// TwinCAT 3 PLC project PLC_1
// ProgramVersion: 3.1.0.4
// libraries:
//   CDS_MemMan, 3.3.2.0 (3S - Smart Software Solutions GmbH)
//   Tc2_Standard, * (Beckhoff Automation GmbH)
//   Tc2_System, * (Beckhoff Automation GmbH)
//   Tc3_Interfaces, * (Beckhoff Automation GmbH)
//   Tc3_Module, * (Beckhoff Automation GmbH)
//   Tc2_Utilities,3.3.0.0,Beckhoff Automation GmbH
// project tree:
//   DUTs/ E_CtrlId.TcDUT (not stored)
//   GVLs/ Global.TcGVL, Io.TcGVL
//   POUs/Alarm/ E_AlmClass.TcDUT, E_AlmState.TcDUT, FB_Alm_Man.TcPOU, T_AlmElement.TcDUT, T_Ctrl_Alm.TcDUT
//   POUs/BaseCtrl/ Base_CmdState.TcGVL, Base_Const.TcGVL, E_Mode.TcDUT, FB_CtrlBase.TcPOU, I_CtrlBase.TcIO, T_Ctrl_CIf.TcDUT, T_Ctrl_Class.TcDUT, T_Ctrl_Class_Alm.TcDUT, T_Ctrl_Class_StateMachine.TcDUT, T_Ctrl_CmdListElement.TcDUT, T_Ctrl_Info.TcDUT, T_Ctrl_IoBool.TcDUT, T_Ctrl_Job.TcDUT, T_Ctrl_SwCfg.TcDUT, T_fbInfo.TcDUT
//   POUs/Controller/Lvl0/CYL/ CYL_CmdState.TcGVL, E_Typ_CYL.TcDUT, FB_CYL.TcPOU, T_Ctrl_SIf_CYL.TcDUT, T_Ctrl_SIf_CYL_Cfg.TcDUT, T_Ctrl_SIf_CYL_Cur.TcDUT, T_Ctrl_SIf_CYL_Ilk.TcDUT (not stored), T_Ctrl_SIf_CYL_In.TcDUT, T_Ctrl_SIf_CYL_Out.TcDUT, T_Ctrl_SIf_CYL_Par.TcDUT
//   POUs/Controller/Lvl2/MOD/ E_Typ_MOD.TcDUT, FB_MOD.TcPOU, MOD_CmdState.TcGVL, T_Ctrl_SIf_MOD.TcDUT, T_Ctrl_SIf_MOD_Cfg.TcDUT (not stored), T_Ctrl_SIf_MOD_Cur.TcDUT, T_Ctrl_SIf_MOD_Ilk.TcDUT, T_Ctrl_SIf_MOD_Par.TcDUT (not stored), T_MOD_RUN_StateMachine.TcDUT (not stored)
//   POUs/Program/ FastPRG_1.TcPOU (not stored), MiddlePRG_1.TcPOU, SlowPRG_1.TcPOU
//   POUs/Utility Functions/ getInBol.TcPOU, getStrInstanceName.TcPOU, setOutBol.TcPOU
//   / Task_Fast.TcTTO, Task_Middle.TcTTO, Task_Slow.TcTTO

CONFIGURATION PLC_1
    RESOURCE PLC ON TwinCAT3
        TASK Task_Fast(INTERVAL := T#10ms, PRIORITY := 5);
        TASK Task_Middle(INTERVAL := T#50000us, PRIORITY := 10);
        TASK Task_Slow(INTERVAL := T#100000us, PRIORITY := 20);
        PROGRAM FastPRG_1 WITH Task_Fast : FastPRG_1;
        PROGRAM MiddlePRG_1 WITH Task_Middle : MiddlePRG_1;
        PROGRAM SlowPRG_1 WITH Task_Slow : SlowPRG_1;
    END_RESOURCE
END_CONFIGURATION

// ---- POUs/Alarm/E_AlmClass.TcDUT
TYPE E_AlmClass :
(
	///no alarm active
	NONE := 0,
	///info
	INFO,
	///warning
	WARNING,
	///tact stop
	TSTOP,
	///stop
	STOP,
	///off
	OFF,
	///Emergency off
	EOFF,
	Max_E_AlmClass
);
END_TYPE

// ---- POUs/Alarm/E_AlmState.TcDUT
TYPE E_AlmState :
(
	///no alarm active
	NONE := 0,
	///alarm clear entry -> set bit1
	CLR := 1,
	///entry resettable alarm ->  set bit2
	RST := 2,
	///entry non resettable alarm ->  set bit2 + bit3
	SET := 3,
	Max_E_AlmState
);
END_TYPE

// ---- POUs/Alarm/T_AlmElement.TcDUT
TYPE T_AlmElement :
STRUCT
	///unique alarm number := 100000*udiMachineNr + intCtrlId*100 + udiAlarmNr
	udiNr: UDINT;
	///additional information - better string???
	dinInfo: DINT;
	///corresponding alarm class
	eClass: E_AlmClass;
	///clear, resetable
	intState: E_AlmState;
	///entry time
	strDTEntry: STRING;
	///from machine (standard = 1)
	udiMachineNr: UDINT;
	///from controller
	intCtrlId: INT;
	///local alarm number
	udiAlarmNr: UDINT;
END_STRUCT
END_TYPE

// ---- POUs/Alarm/T_Ctrl_Alm.TcDUT
TYPE T_Ctrl_Alm :
STRUCT
	///alarm flag array
	bol: BOOL;
	eAlmClass: E_AlmClass;
	strText: STRING;
END_STRUCT
END_TYPE

// ---- POUs/BaseCtrl/E_Mode.TcDUT
{attribute 'qualified_only' := ''}
TYPE E_Mode :
(
	INITIALIZED := 0,
	AUTO := 10,
	SEMI := 11,
	MANU := 12
);
END_TYPE

// ---- POUs/BaseCtrl/T_Ctrl_CIf.TcDUT
TYPE T_Ctrl_CIf :
STRUCT
	Job: T_Ctrl_Job;
	Info: T_Ctrl_Info;
	SwCfg: T_Ctrl_SwCfg;
END_STRUCT
END_TYPE

// ---- POUs/BaseCtrl/T_Ctrl_Class.TcDUT
TYPE T_Ctrl_Class :
STRUCT
	///local test flag to supress cyclic run (for debugging after init)
	bolActivate: BOOL;
	intCmd: INT;
	intCmdLast: INT;
	eModeHistory: E_Mode;
	///local flag mode change detected
	bolChangeBackToAUTO: BOOL;
	StateMachine: T_Ctrl_Class_StateMachine;
	Alarm: T_Ctrl_Class_Alm;
	FUBInfo: T_fbInfo;
END_STRUCT
END_TYPE

// ---- POUs/BaseCtrl/T_Ctrl_Class_Alm.TcDUT
TYPE T_Ctrl_Class_Alm :
STRUCT
	bolResetOk: BOOL;
	///flag positive check me alarm from child
	bolfp: BOOL;
	///local activ alarm class of parent ctrl
	eParent_ActivAlmClass: E_AlmClass;
	///highest local activ alarm class
	eActivAlmClass: E_AlmClass;
END_STRUCT
END_TYPE

// ---- POUs/BaseCtrl/T_Ctrl_Class_StateMachine.TcDUT
TYPE T_Ctrl_Class_StateMachine :
STRUCT
	///actual state
	intState: INT;
	///state of last cycle
	intStateLastCycle: INT;
	///save history backup p.e. in ERROR state
	intStateHistory: INT;
	///set state for next cycle
	intStateNext: INT;
	///[ms] to simulate state in SINGLE_ANSWER
	udiStateSimSetTime_ms: UDINT := 1000;
	///[ms] time in one state
	udiTimeInState_ms: UDINT;
END_STRUCT
END_TYPE

// ---- POUs/BaseCtrl/T_Ctrl_CmdListElement.TcDUT
TYPE T_Ctrl_CmdListElement :
STRUCT
	///command implemented in controller
	intCmd: INT;
	///command is available info for UI
	bolAvailable: BOOL;
	
	// Name of command. Important for UI.
	strName: STRING;
END_STRUCT
END_TYPE

// ---- POUs/BaseCtrl/T_Ctrl_Info.TcDUT
TYPE T_Ctrl_Info :
STRUCT
	///name of controller instance
	strName: STRING(80);
	///class of controller
	strType: STRING(80);
	///unique controller instance identification number
	intCtrlId: INT;
	///unique identification number of parent controller instance
	intParentCtrlId: INT;
	///all inputs valid -> init done
	bolInitDone: BOOL;
	///Childs
	p_afbChild: ARRAY[0..Base_Const.cMaxNrOfChilds] OF POINTER TO BYTE;
	///common interface array of childs
	p_aCIf: ARRAY[0..Base_Const.cMaxNrOfChilds] OF POINTER TO T_Ctrl_CIf;
END_STRUCT
END_TYPE

// ---- POUs/BaseCtrl/T_Ctrl_IoBool.TcDUT
TYPE T_Ctrl_IoBool :
STRUCT
	///mapped io variable to hardware
	map: BOOL;
	///shows the state of (input: mapped, output: set by programm respectiv at the moment one cycle later evtl. from the forcing if forcing active) -> necessary for what?
	state: BOOL;
	///variabel to/ from program
	intern: BOOL;
	///variabel set from UI
	force: BOOL;
	///enable force of single io-datapoint
	EnForce: BOOL;
END_STRUCT
END_TYPE

// ---- POUs/BaseCtrl/T_Ctrl_Job.TcDUT
TYPE T_Ctrl_Job :
STRUCT
	///mode if mode = AUTO -> ACmd will be used, otherwise the MCmd channel is open
	eMode: E_Mode;
	///automatic command from parent ctrl
	intACmd: INT;
	///manual command from UI p.e.
	intMCmd: INT;
	///active cmd
	strCmd: STRING;
	///active state
	intState: INT;
	strState: STRING;
	///if used - show substates for debugging
	strSubState: STRING;
	///event channel to signal special events to parent parallel to status
	intEvt: INT;
	///reset all alarms
	bolAlmReset: BOOL;
	///activate io-forcing
	bolIoForce: BOOL;
	///overwrite suspend all interlocks (for debugging/testing)
	bolIlkOverwrite: BOOL;
	///activ alarm class of parent ctrl
	eParent_ActivAlmClass: E_AlmClass;
	///activ alarm class of me ctrl
	eMe_ActivAlmClass: E_AlmClass;
	///list of all implemented commands
	aCmdList: ARRAY[0..cMaxCmdPerCtrl] OF T_Ctrl_CmdListElement;
END_STRUCT
END_TYPE

// ---- POUs/BaseCtrl/T_Ctrl_SwCfg.TcDUT
TYPE T_Ctrl_SwCfg :
STRUCT
	///hardware/controller exists
	bolExist: BOOL;
	///enable statemachine
	bolEnable: BOOL;
	///set controller in simulation(statemachine active, io local simulated)
	bolSimulation: BOOL;
END_STRUCT
END_TYPE

// ---- POUs/BaseCtrl/T_fbInfo.TcDUT
TYPE T_fbInfo :
STRUCT
	udiSample_ms: UDINT;
END_STRUCT
END_TYPE

// ---- POUs/Controller/Lvl0/CYL/E_Typ_CYL.TcDUT
TYPE E_Typ_CYL :
(
	///bistabile and two feedback sensors
	Valve2_Sensor2 := 0,
	///bistabile and extended feedback sensors	
	Valve2_SensorExtended,
	///bistabile and retracted feedback sensors	
	Valve2_SensorRetracted,
	///bistabile and no feedback sensors
	Valve2_Sensor0,
	///monostabile and 2 feedback sensors	
	Valve1_Sensor2,
	///monostabile and extended feedback sensors	
	Valve1_SensorExtended,
	///monostabile and retracted feedback sensor
	Valve1_SensorRetracted,
	///monostabile and no feedback sensors
	Valve1_Sensor0,
	Max_E_Typ_CYL
);
END_TYPE

// ---- POUs/Controller/Lvl0/CYL/T_Ctrl_SIf_CYL.TcDUT
TYPE T_Ctrl_SIf_CYL :
STRUCT
	///configuration
	Cfg: T_Ctrl_SIf_CYL_Cfg;
	///parameter
	Par: T_Ctrl_SIf_CYL_Par;
	///current values
	Cur: T_Ctrl_SIf_CYL_Cur;
	///io input
	In: T_Ctrl_SIf_CYL_In;
	///io output
	Out: T_Ctrl_SIf_CYL_Out;
	///alarm number used in this controller
	Alm: ARRAY[1..6] OF T_Ctrl_Alm;
	///interlock of output/movements
	Ilk: T_Ctrl_SIf_CYL_Ilk;
END_STRUCT
END_TYPE

// ---- POUs/Controller/Lvl0/CYL/T_Ctrl_SIf_CYL_Cfg.TcDUT
TYPE T_Ctrl_SIf_CYL_Cfg :
STRUCT
	eTyp: E_Typ_CYL;
END_STRUCT
END_TYPE

// ---- POUs/Controller/Lvl0/CYL/T_Ctrl_SIf_CYL_Cur.TcDUT
TYPE T_Ctrl_SIf_CYL_Cur :
STRUCT
	///[ms] time last movement to retract
	udiMoveTimeRetract: UDINT;
	///[ms] time last movement to extend
	udiMoveTimeExtend: UDINT;
END_STRUCT
END_TYPE

// ---- POUs/Controller/Lvl0/CYL/T_Ctrl_SIf_CYL_In.TcDUT
TYPE T_Ctrl_SIf_CYL_In :
STRUCT
	///sensor feedback position extended reached
	bolExtended: T_Ctrl_IoBool;
	///sensor feedback position retracted reached
	bolRetracted: T_Ctrl_IoBool;
END_STRUCT
END_TYPE

// ---- POUs/Controller/Lvl0/CYL/T_Ctrl_SIf_CYL_Out.TcDUT
TYPE T_Ctrl_SIf_CYL_Out :
STRUCT
	///switch valve retract
	bolRetract: T_Ctrl_IoBool;
	///switch valve extend
	bolExtend: T_Ctrl_IoBool;
END_STRUCT
END_TYPE

// ---- POUs/Controller/Lvl0/CYL/T_Ctrl_SIf_CYL_Par.TcDUT
TYPE T_Ctrl_SIf_CYL_Par :
STRUCT
	///[ms] until failure to long time for extend
	udiExtendTime_ms: UDINT;
	///[ms] until failure to long time for retract
	udiRetractTime_ms: UDINT;
	///[ms] simulation time for extend or /2 of timeout time?
	udiSimExtendTime_ms: UDINT;
	///[ms] simulation time for retract or /2 of timeout time?
	udiSimRetractTime_ms: UDINT;
END_STRUCT
END_TYPE

// ---- POUs/Controller/Lvl2/MOD/E_Typ_MOD.TcDUT
TYPE E_Typ_MOD :
(
	///no usage until yet
	Default := 0,
	Max_E_Typ_CYL
);
END_TYPE

// ---- POUs/Controller/Lvl2/MOD/T_Ctrl_SIf_MOD.TcDUT
TYPE T_Ctrl_SIf_MOD :
STRUCT
	///configuration
	Cfg: T_Ctrl_SIf_MOD_Cfg;
	///parameter
	Par: T_Ctrl_SIf_MOD_Par;
	///current values
	Cur: T_Ctrl_SIf_MOD_Cur;
	///In: T_Ctrl_SIf_MOD_In;
	///Out: T_Ctrl_SIf_MOD_Out;
	Alm: ARRAY[1..6] OF T_Ctrl_Alm;
END_STRUCT
END_TYPE

// ---- POUs/Controller/Lvl2/MOD/T_Ctrl_SIf_MOD_Cur.TcDUT
TYPE T_Ctrl_SIf_MOD_Cur :
STRUCT
	///[ms] time last cycle
	udiCycleTime_ms: UDINT;
END_STRUCT
END_TYPE

// ---- POUs/Controller/Lvl2/MOD/T_Ctrl_SIf_MOD_Ilk.TcDUT
TYPE T_Ctrl_SIf_MOD_Ilk :
STRUCT
	///interlock retraction of cylinder
	bolRetract: BOOL;
	///interlock extend of cylinder
	bolExtend: BOOL;
END_STRUCT
END_TYPE

// ---- GVLs/Global.TcGVL
VAR_GLOBAL
	g_a_pCtrlInst: ARRAY[0..E_CtrlId.E_CtrlIdMax] OF POINTER TO fb_CtrlBase;
	g_a_pCtrlCIf: ARRAY[0..E_CtrlId.E_CtrlIdMax] OF POINTER TO T_Ctrl_CIf;
	g_fbAlm_Man: FB_Alm_Man;
END_VAR

// ---- GVLs/Io.TcGVL
VAR_GLOBAL
	///input fb instance Cyl_AB position retract normally open
	In_bolCyl_AB_Retracted_NO: BOOL;
	///input fb instance Cyl_AB position extend normally closed
	In_bolCyl_AB_Extended_NC: BOOL;
	///output fb instance Cyl_AB valve retract
	Out_bolCyl_AB_Retract: BOOL;
	///output fb instance Cyl_AB valve extend
	Out_bolCyl_AB_Extend: BOOL;
END_VAR

// ---- POUs/BaseCtrl/Base_CmdState.TcGVL
VAR_GLOBAL CONSTANT
	///ctrl commands definitions
	///general commands 2-200 - every command has to be a even number
	cCMD_DONE: INT := -1;
	cCMD_INITIALIZED: INT := 0;
	cCMD_PON: INT := 2;
	cCMD_EOFF: INT := 4;
	cCMD_OFF: INT := 6;
	cCMD_INIT: INT := 8;
	cCMD_RUN: INT := 10;
	cCMD_STOP: INT := 12;
	cCMD_TSTOP: INT := 14;
	///ctrl states definitions
	cSTA_DONE: INT := cCMD_DONE;
	cSTA_INITIALIZED: INT := cCMD_INITIALIZED;
	cSTA_PONBusy: INT := 1;
	cSTA_PON: INT := cCMD_PON;
	cSTA_EOFFBusy: INT := 3;
	cSTA_EOFF: INT := cCMD_EOFF;
	cSTA_OFFBusy: INT := 5;
	cSTA_OFF: INT := cCMD_OFF;
	cSTA_INITBusy: INT := 7;
	cSTA_INIT: INT := cCMD_INIT;
	cSTA_RUNBusy: INT := 9;
	cSTA_RUN: INT := cCMD_RUN;
	cSTA_STOPBusy: INT := 11;
	cSTA_STOP: INT := cCMD_STOP;
	cSTA_TSTOPBusy: INT := 13;
	cSTA_TSTOP: INT := cCMD_TSTOP;
	///special states without corresponding cmd
	cSTA_ERROR: INT := 150;
	cSTA_ERRORQuit: INT := 151;
	cSTA_SINGLE_ANSWER: INT := 152;
END_VAR

// ---- POUs/BaseCtrl/Base_Const.TcGVL
VAR_GLOBAL CONSTANT
	///number of child access possible in one controller class
	cMaxNrOfChilds: UINT := 10;
	///maximal number of commands implemented in one controller class
	cMaxCmdPerCtrl: UINT := 15;
	///maximal number of commands implemented in one controller class
	cMaxBaseCmdState: UINT := 200;
END_VAR

// ---- POUs/Controller/Lvl0/CYL/CYL_CmdState.TcGVL
VAR_GLOBAL CONSTANT
	///ctrl commands definitions
	///specific commands >200 - every command has to be a even number
	cCMD_RETRACT: INT := 202;
	cCMD_EXTEND: INT := 204;
	///ctrl specific states definitions
	cSTA_RETRACTBusy: INT := 201;
	cSTA_RETRACT: INT := cCMD_RETRACT;
	cSTA_EXTENDBusy: INT := 203;
	cSTA_EXTEND: INT := cCMD_EXTEND;
END_VAR

// ---- POUs/Controller/Lvl2/MOD/MOD_CmdState.TcGVL
VAR_GLOBAL CONSTANT
	///ctrl commands definitions
	///specific commands >200 - every command has to be a even number
	///ctrl specific states definitions
	cSTA_VER_Up: INT := 201;
	cSTA_VER_Down: INT := 202;
	cSTA_WAIT_Pick: INT := 203;
	cSTA_HOR_MoveToPlace: INT := 204;
	cSTA_HOR_MoveToPick: INT := 205;
	cSTA_Finished: INT := 206;
END_VAR

// ---- POUs/BaseCtrl/I_CtrlBase.TcIO
INTERFACE I_CtrlBase

METHOD iniCtrlArray : BOOL
VAR_INPUT
	p_pCtrlArray: POINTER TO POINTER TO fb_CtrlBase;
	intCtrlID: INT;
END_VAR
END_METHOD

METHOD getCtrlCIf : POINTER TO T_Ctrl_CIf
END_METHOD

END_INTERFACE

// ---- POUs/Program/MiddlePRG_1.TcPOU
PROGRAM MiddlePRG_1
VAR
	bolPlcStartupDone: BOOL := FALSE;
	bolHostInitDone : BOOL := FALSE;
	bolInitDone : BOOL := FALSE;
	fbCyl_AB: FB_CYL;
	fbMOD_2: FB_MOD;
	fbVER_2: FB_CYL;
	fbHOR_2: FB_CYL;
END_VAR

(*__________________________________________________________________________________________________
¦	
¦	Vistaprint Schweiz GmbH
¦	CH - 8401 Winterthur
¦
¦	www.vistaprint.ch - info@vistaprint.ch
¦___________________________________________________________________________________________________

Function desription:
call of all controller (FUB) for the middel task class inclusiv alarm handler.


History:
Version		Date			Author		Comment
---------------------------------------------------------------------------------------------------
0.00.1		02.05.2013		AVME/KVO	Start history


___________________________________________________________________________________________________*)

// -----------------------------------------------------------------------------------------------
// Initialize the PLC Parameter and check the PLC health
// -----------------------------------------------------------------------------------------------
IF (NOT bolPlcStartupDone) THEN
	bolPlcStartupDone := TRUE;	
END_IF
// -----------------------------------------------------------------------------------------------


// -----------------------------------------------------------------------------------------------
// The host system is downloading all parameter at startup. 
// bolPlcStartupDone will be set to true after the Host is done with the initialization
// -----------------------------------------------------------------------------------------------
IF (bolPlcStartupDone AND (NOT bolHostInitDone) AND NOT bolInitDone) THEN
	bolHostInitDone := TRUE;
END_IF
// -----------------------------------------------------------------------------------------------


// -----------------------------------------------------------------------------------------------
// Start PLC code initialization
// -----------------------------------------------------------------------------------------------
IF NOT bolInitDone AND bolPlcStartupDone AND bolHostInitDone THEN
	
	// init
	fbCyl_AB.iniCtrlArray(ADR(g_a_pCtrlInst),E_CtrlId.CYL_VER1);     	// init and entry fb_instance in global fb pointer array
	g_a_pCtrlCIf[E_CtrlId.CYL_VER1] := fbCyl_AB.getCtrlCIf();    // get adr of ctrl interface struct
	
	// init module example
	// Lvl0
	fbHOR_2.iniCtrlArray(ADR(g_a_pCtrlInst),E_CtrlId.HOR_2); // init and entry fb_instance in global fb pointer array
	g_a_pCtrlCIf[E_CtrlId.HOR_2] := fbHOR_2.getCtrlCIf();    // get adr of ctrl interface struct
	
	fbVER_2.iniCtrlArray(ADR(g_a_pCtrlInst),E_CtrlId.VER_2); // init and entry fb_instance in global fb pointer array
	g_a_pCtrlCIf[E_CtrlId.VER_2] := fbVER_2.getCtrlCIf();    // get adr of ctrl interface struct
	
	//Lvl2
	fbMOD_2.iniCtrlArray(ADR(g_a_pCtrlInst),E_CtrlId.MOD_2); // init and entry fb_instance in global fb pointer array
	g_a_pCtrlCIf[E_CtrlId.MOD_2] := fbMOD_2.getCtrlCIf();    // get adr of ctrl interface struct
	
	// add childs
	fbMOD_2.p_fbHOR := g_a_pCtrlInst[E_CtrlId.HOR_2];
	fbMOD_2.p_fbVER := g_a_pCtrlInst[E_CtrlId.VER_2];

	// add childs
	fbMOD_2.p_fbHOR := g_a_pCtrlInst[E_CtrlId.HOR_2];
	fbMOD_2.p_fbVER := g_a_pCtrlInst[E_CtrlId.VER_2];

	bolInitDone := TRUE;
END_IF
// -----------------------------------------------------------------------------------------------



// -----------------------------------------------------------------------------------------------
// Normal Run mode after all the initialization is done
// -----------------------------------------------------------------------------------------------
IF (bolInitDone AND bolPlcStartupDone AND bolHostInitDone) THEN
	
	//****************************************************************************************************
	// cyclic controller calls
	//****************************************************************************************************
	fbCyl_AB.In_bolRetracted := In_bolCyl_AB_Retracted_NO;
	fbCyl_AB.In_bolExtended := (NOT In_bolCyl_AB_Extended_NC);
	fbCyl_AB();
	Out_bolCyl_AB_Retract := fbCyl_AB.Out_bolRetract;
	Out_bolCyl_AB_Extend := fbCyl_AB.Out_bolExtend;

	// Modul example
	// ----------------------------------------------------------------------------------------------------------------------------
	// modul controller MOD_2 with childs
	fbMOD_2();
	fbVER_2();
	fbHOR_2();

	
END_IF
// -----------------------------------------------------------------------------------------------

END_PROGRAM

// ---- POUs/Controller/Lvl0/CYL/FB_CYL.TcPOU
FUNCTION_BLOCK FB_CYL EXTENDS FB_CtrlBase

VAR_INPUT
	In_bolRetracted: BOOL;
	In_bolExtended: BOOL;
END_VAR
VAR_OUTPUT
	Out_bolRetract: BOOL;
	Out_bolExtend: BOOL;
END_VAR

VAR
	/// Specific interface struct for public access
	SIf: T_Ctrl_SIf_CYL;
	
END_VAR

(*__________________________________________________________________________________________________
¦	
¦	Vistaprint Schweiz GmbH
¦	CH - 8401 Winterthur
¦
¦	www.vistaprint.ch - info@vistaprint.ch
¦___________________________________________________________________________________________________

Function desription:
Basic controller implementation. This Controller should be the base father controller for all in the
feature implemented ctontroller classes.


History:
Version		Date			Author		Comment
---------------------------------------------------------------------------------------------------
0.00.1		25.04.2013		AVME/KVO	Start history


___________________________________________________________________________________________________*)


IF (me.bolActivate) THEN // cyclic call enabled
	IF (CIf.Info.bolInitDone=FALSE) THEN // first cycle -> init
		CtrlInit();
		CIf.Info.bolInitDone := TRUE;
	ELSE
		CycleStartDuty();
	
		Always();
		
		StateMachine();
		
		CycleEndDuty();
	END_IF
END_IF;

METHOD FB_init : BOOL
VAR_INPUT
	///if TRUE, the retain variables are initialized (warm start / cold start)
	bInitRetains: BOOL;
	///if TRUE, the instance afterwards gets moved into the copy code (online change)
	bInCopyCode: BOOL;
END_VAR
VAR
	udiTaskCnt: UDINT;
	ii: UINT;
END_VAR
//------------------------------------------------------------------------------------------------------------------------
// to manually change in new FUB implementation!!!
// define valid commands for this controller
FOR ii:= 0 TO (SIZEOF(CIf.Job.aCmdList)/SIZEOF(CIf.Job.aCmdList[0])-1) BY 1 DO
	IF (CIf.Job.aCmdList[ii].intCmd=cCMD_INITIALIZED) THEN
		// found first empty array element
		EXIT;
	END_IF
END_FOR
CIf.Job.aCmdList[ii].intCmd := cCMD_STOP;
CIf.Job.aCmdList[ii].strName := 'Stop'; 
CIf.Job.aCmdList[ii].bolAvailable := TRUE;
ii := ii +1;
CIf.Job.aCmdList[ii].intCmd := cCMD_RETRACT;
CIf.Job.aCmdList[ii].strName := 'Retract';
CIf.Job.aCmdList[ii].bolAvailable := TRUE;
ii := ii +1;
CIf.Job.aCmdList[ii].intCmd := cCMD_EXTEND; // for test simulation single answer
CIf.Job.aCmdList[ii].strName := 'Extend';
CIf.Job.aCmdList[ii].bolAvailable := TRUE;

// set name of class/typ
CIf.Info.strType := 'FB_CYL'; 

// set alarm class
SIf.Alm[1].eAlmClass := E_AlmClass.EOFF;
//SIf.Alm[1].strAlarm := 'Alarmtext 1';
SIf.Alm[2].eAlmClass := E_AlmClass.OFF;
SIf.Alm[3].eAlmClass := E_AlmClass.STOP;
SIf.Alm[4].eAlmClass := E_AlmClass.TSTOP;
SIf.Alm[5].eAlmClass := E_AlmClass.INFO;
SIf.Alm[6].eAlmClass := E_AlmClass.WARNING;

//*******************************************************************************
// initial values
//*******************************************************************************

// software configuration
CIf.SwCfg.bolExist := TRUE;
CIf.SwCfg.bolSimulation := TRUE;

// parmeter
SIf.Par.udiExtendTime_ms := 10000;
SIf.Par.udiRetractTime_ms := 8000;
SIf.Par.udiSimExtendTime_ms := SIf.Par.udiExtendTime_ms/2;	
SIf.Par.udiSimRetractTime_ms := SIf.Par.udiRetractTime_ms/2;
END_METHOD

METHOD PROTECTED IoInBridge : BOOL
// digitale and analoge inputs read from hardware or forcing
SIf.In.bolExtended.map := THIS^.In_bolExtended;
SIf.In.bolRetracted.map := THIS^.In_bolRetracted;

IF (CIf.SwCfg.bolSimulation = FALSE) THEN
	getInBol(CIf.Job.bolIoForce,ADR(SIf.In.bolExtended));
	getInBol(CIf.Job.bolIoForce,ADR(SIf.In.bolRetracted));
	//ctrl.In.bol_PosSwitchBasicDefTyp.intern := getInBol(ctrl.ifc.Job.bol_Force ,ADR(ctrl.In.bol_PosSwitchBasicDefTyp);
ELSE
	//simulation of global IO
END_IF
END_METHOD

METHOD PROTECTED IoOutBridge : BOOL
VAR
	bolSwitchValvesOff: BOOL;
END_VAR
// digitale and analoge inputs read from hardware or forcing
IF (CIf.SwCfg.bolSimulation = FALSE) THEN
	// check interlocks to prevent damages
	IF (CIf.Job.bolIlkOverwrite=FALSE) THEN
		bolSwitchValvesOff := FALSE;
		
		IF (SIf.Ilk.bolExtend=FALSE) THEN
			setOutBol(CIf.Job.bolIoForce ,ADR(SIf.Out.bolExtend));
		ELSE
			// switch off?
			IF (SIf.Cfg.eTyp = E_Typ_CYL.Valve1_Sensor0) OR (SIf.Cfg.eTyp = E_Typ_CYL.Valve1_Sensor2) 
				OR (SIf.Cfg.eTyp = E_Typ_CYL.Valve1_SensorExtended) OR (SIf.Cfg.eTyp = E_Typ_CYL.Valve1_SensorRetracted) THEN
				// monostabil valve -> do nothing
			ELSE
				// bistable valve ->  switch both off
				bolSwitchValvesOff := TRUE;
			END_IF
		END_IF
		
		IF (SIf.Ilk.bolRetract=FALSE) THEN
			setOutBol(CIf.Job.bolIoForce ,ADR(SIf.Out.bolRetract));
		ELSE
			// switch off?
			IF (SIf.Cfg.eTyp = E_Typ_CYL.Valve1_Sensor0) OR (SIf.Cfg.eTyp = E_Typ_CYL.Valve1_Sensor2) 
				OR (SIf.Cfg.eTyp = E_Typ_CYL.Valve1_SensorExtended) OR (SIf.Cfg.eTyp = E_Typ_CYL.Valve1_SensorRetracted) THEN
				// monostabil valve -> do nothing
				;
			ELSE
				// bistable valve -> switch both off
				bolSwitchValvesOff := TRUE;
			END_IF
		END_IF
		
		// bistable valve -> switch both off
		IF (bolSwitchValvesOff) THEN
			SIf.Out.bolExtend.map := FALSE;
			SIf.Out.bolRetract.map := FALSE;
		END_IF
		
	END_IF
END_IF
END_METHOD

METHOD PROTECTED StateMachine : BOOL
SUPER^.StateMachine();

// main statemachine of base controller
CASE me.StateMachine.intState OF
    cSTA_RETRACTBusy: 
        THIS^.sta_RETRACTBusy();
    cSTA_RETRACT: 
        THIS^.sta_RETRACT();
    cSTA_EXTENDBusy: 
        THIS^.sta_EXTENDBusy();
    cSTA_EXTEND: 
        THIS^.sta_EXTEND();
END_CASE;
END_METHOD

METHOD PROTECTED sta_ERROR : BOOL
// state implemetation
//--------------------------------------------------------------------------------------
// Entry action
	IF (me.StateMachine.intState<>me.StateMachine.intStateHistory) THEN
		me.StateMachine.intStateHistory := me.StateMachine.intStateLastCycle; // -> possibillity to go back to state before error
		me.StateMachine.intStateLastCycle := me.StateMachine.intState;
		
	END_IF


//--------------------------------------------------------------------------------------
// Cyclic action
	IF (me.StateMachine.intState=me.StateMachine.intStateLastCycle) THEN
		
		;
		
		
		// State Change Condition
		IF (CIf.Job.bolAlmReset = TRUE) THEN
			me.StateMachine.intStateNext := cSTA_ERRORQuit;
		END_IF
	END_IF




//--------------------------------------------------------------------------------------
// Exit action
	IF (me.StateMachine.intState<>me.StateMachine.intStateNext) THEN
		;
	END_IF
END_METHOD

METHOD PROTECTED sta_ERRORQuit : BOOL
// state implemetation
//--------------------------------------------------------------------------------------
// Entry action
	IF (me.StateMachine.intState<>me.StateMachine.intStateLastCycle) THEN
		me.StateMachine.intStateLastCycle := me.StateMachine.intState;
		
	END_IF


//--------------------------------------------------------------------------------------
// Cyclic action
	IF (me.StateMachine.intState=me.StateMachine.intStateLastCycle) THEN
		
		;
		// evtl. wait time if reset of device is necessary and then decide to go to states or ERROR state
		IF (CIf.Job.bolAlmReset = TRUE) THEN
			CIf.Job.eMe_ActivAlmClass := E_AlmClass.NONE; // reset feedback channel for parent
			CIf.Job.bolAlmReset := FALSE;
		END_IF
		
		// State Change Condition
		IF (CIf.Job.bolAlmReset = FALSE) THEN
			IF (me.StateMachine.intStateHistory<=cSTA_PON) THEN
				me.StateMachine.intStateNext := cSTA_PONBusy;
			ELSIF(me.intCmd=cCMD_OFF) THEN
				me.StateMachine.intStateNext := cSTA_OFFBusy;
			ELSIF(me.intCmd=cCMD_STOP) THEN
				me.StateMachine.intStateNext := cSTA_STOPBusy;
			ELSIF(me.intCmd=cCMD_RETRACT) THEN
				me.StateMachine.intStateNext := cSTA_RETRACTBusy;
			ELSIF(me.intCmd=cCMD_EXTEND) THEN
				me.StateMachine.intStateNext := cSTA_EXTENDBusy;
			END_IF
		END_IF
	END_IF




//--------------------------------------------------------------------------------------
// Exit action
	IF (me.StateMachine.intState<>me.StateMachine.intStateNext) THEN
		;
	END_IF
END_METHOD

METHOD PROTECTED sta_EXTENDBusy : BOOL
// state implemetation
//--------------------------------------------------------------------------------------
// Entry action
	IF (me.StateMachine.intState<>me.StateMachine.intStateLastCycle) THEN
		me.StateMachine.intStateLastCycle := me.StateMachine.intState;

		fbSimulationTimer.IN := FALSE;
		fbSimulationTimer.PT := UDINT_TO_TIME(SIf.Par.udiSimExtendTime_ms);
		fbSimulationTimer(); // set time/reset timer
		fbSimulationTimer.IN := TRUE; // start timer
	END_IF


//--------------------------------------------------------------------------------------
// Cyclic action
	IF (me.StateMachine.intState=me.StateMachine.intStateLastCycle) THEN

		// Simulation
		IF (CIf.SwCfg.bolSimulation) THEN
			fbSimulationTimer(); // simulation time
			IF (fbSimulationTimer.Q) THEN
				SIf.In.bolExtended.intern := TRUE;
				SIf.In.bolRetracted.intern := FALSE;
			END_IF
		END_IF
		
		//no change action
		SIf.Out.bolExtend.intern := TRUE;
		SIf.Out.bolRetract.intern := FALSE;
		
		
		// State Change Condition
		IF (me.StateMachine.udiTimeInState_ms>SIf.Par.udiExtendTime_ms) THEN
			IF (SIf.In.bolRetracted.intern) THEN
				// sensor retract always on cylinder
				g_fbAlm_Man.setAlarm(CIf.Info.intCtrlId,1,777,ADR(SIf.Alm),E_AlmState.RST,CIf.Job.eMe_ActivAlmClass);
			ELSE
				// timeout extend cylinder
				g_fbAlm_Man.setAlarm(CIf.Info.intCtrlId,2,0,ADR(SIf.Alm),E_AlmState.RST,CIf.Job.eMe_ActivAlmClass);
			END_IF
			me.StateMachine.intStateNext :=  cSTA_ERROR;
		ELSIF (SIf.In.bolExtended.intern) AND (SIf.In.bolRetracted.intern=FALSE) THEN
			me.StateMachine.intStateNext := cSTA_EXTEND;
		ELSIF(me.intCmd=cCMD_OFF) THEN
			me.StateMachine.intStateNext := cSTA_OFFBusy;
		ELSIF(me.intCmd=cCMD_STOP) THEN
			me.StateMachine.intStateNext := cSTA_STOPBusy;
		ELSIF(me.intCmd=cCMD_RETRACT) THEN
			me.StateMachine.intStateNext := cSTA_RETRACTBusy;
		END_IF
	END_IF




//--------------------------------------------------------------------------------------
// Exit action
	IF (me.StateMachine.intState<>me.StateMachine.intStateNext) THEN
		SIf.Cur.udiMoveTimeExtend := me.StateMachine.udiTimeInState_ms;
	END_IF
END_METHOD

METHOD PROTECTED sta_EXTEND : BOOL
// state implemetation
//--------------------------------------------------------------------------------------
// Entry action
	IF (me.StateMachine.intState<>me.StateMachine.intStateLastCycle) THEN
		me.StateMachine.intStateLastCycle := me.StateMachine.intState;

	END_IF


//--------------------------------------------------------------------------------------
// Cyclic action
	IF (me.StateMachine.intState=me.StateMachine.intStateLastCycle) THEN

		// Simulation
		IF (CIf.SwCfg.bolSimulation) THEN
			;
		END_IF
		
		// State Change Condition
		IF (SIf.In.bolRetracted.intern) THEN
			// sensor retract always on cylinder
			me.StateMachine.intStateNext :=  cSTA_ERROR;
		ELSIF (SIf.In.bolExtended.intern = FALSE) THEN // wait time until error?
			me.StateMachine.intStateNext := cSTA_EXTENDBusy;
		ELSIF(me.intCmd=cCMD_OFF) THEN
			me.StateMachine.intStateNext := cSTA_OFFBusy;
		ELSIF(me.intCmd=cCMD_STOP) THEN
			me.StateMachine.intStateNext := cSTA_STOPBusy;
		ELSIF(me.intCmd=cCMD_RETRACT) THEN
			me.StateMachine.intStateNext := cSTA_RETRACTBusy;
		END_IF
	END_IF




//--------------------------------------------------------------------------------------
// Exit action
	IF (me.StateMachine.intState<>me.StateMachine.intStateNext) THEN
		;
	END_IF
END_METHOD

METHOD PROTECTED sta_RETRACT : BOOL
// state implemetation
//--------------------------------------------------------------------------------------
// Entry action
	IF (me.StateMachine.intState<>me.StateMachine.intStateLastCycle) THEN
		me.StateMachine.intStateLastCycle := me.StateMachine.intState;

	END_IF


//--------------------------------------------------------------------------------------
// Cyclic action
	IF (me.StateMachine.intState=me.StateMachine.intStateLastCycle) THEN

		// Simulation
		IF (CIf.SwCfg.bolSimulation) THEN
			;
		END_IF
		
		// State Change Condition
		IF (SIf.In.bolExtended.intern) THEN
			// sensor retract always on cylinder
			me.StateMachine.intStateNext :=  cSTA_ERROR;
		ELSIF (SIf.In.bolRetracted.intern = FALSE) THEN // wait time until error?
			me.StateMachine.intStateNext := cSTA_RETRACTBusy;
		ELSIF(me.intCmd=cCMD_OFF) THEN
			me.StateMachine.intStateNext := cSTA_OFFBusy;
		ELSIF(me.intCmd=cCMD_STOP) THEN
			me.StateMachine.intStateNext := cSTA_STOPBusy;
		ELSIF(me.intCmd=cCMD_EXTEND) THEN
			me.StateMachine.intStateNext := cSTA_EXTENDBusy;
		END_IF
	END_IF




//--------------------------------------------------------------------------------------
// Exit action
	IF (me.StateMachine.intState<>me.StateMachine.intStateNext) THEN
		;
	END_IF
END_METHOD

METHOD PROTECTED sta_RETRACTBusy : BOOL
// state implemetation
//--------------------------------------------------------------------------------------
// Entry action
	IF (me.StateMachine.intState<>me.StateMachine.intStateLastCycle) THEN
		me.StateMachine.intStateLastCycle := me.StateMachine.intState;
		
		SIf.Out.bolExtend.intern := FALSE;
		SIf.Out.bolRetract.intern := TRUE;
		
		fbSimulationTimer.IN := FALSE;
		fbSimulationTimer.PT := UDINT_TO_TIME(SIf.Par.udiSimRetractTime_ms);
		fbSimulationTimer(); // set time/reset timer
		fbSimulationTimer.IN := TRUE; // start timer
	END_IF


//--------------------------------------------------------------------------------------
// Cyclic action
	IF (me.StateMachine.intState=me.StateMachine.intStateLastCycle) THEN

		// Simulation
		IF (CIf.SwCfg.bolSimulation) THEN
			fbSimulationTimer(); // simulation time
			IF (fbSimulationTimer.Q) THEN
				SIf.In.bolRetracted.intern := TRUE;
				SIf.In.bolExtended.intern := FALSE;
			END_IF
		END_IF
		
		// State Change Condition
		IF (me.StateMachine.udiTimeInState_ms>SIf.Par.udiRetractTime_ms) THEN
			IF (SIf.In.bolExtended.intern) THEN
				// sensor retract always on cylinder
				g_fbAlm_Man.setAlarm(CIf.Info.intCtrlId,3,0,ADR(SIf.Alm),E_AlmState.RST,CIf.Job.eMe_ActivAlmClass);
			ELSE
				// timeout extend cylinder
				g_fbAlm_Man.setAlarm(CIf.Info.intCtrlId,4,0,ADR(SIf.Alm),E_AlmState.RST,CIf.Job.eMe_ActivAlmClass);
			END_IF
			me.StateMachine.intStateNext :=  cSTA_ERROR;
		ELSIF (SIf.In.bolRetracted.intern) AND(SIf.In.bolExtended.intern=FALSE) THEN
			me.StateMachine.intStateNext := cSTA_RETRACT;
		ELSIF(me.intCmd=cCMD_OFF) THEN
			me.StateMachine.intStateNext := cSTA_OFFBusy;
		ELSIF(me.intCmd=cCMD_STOP) THEN
			me.StateMachine.intStateNext := cSTA_STOPBusy;
		ELSIF(me.intCmd=cCMD_EXTEND) THEN
			me.StateMachine.intStateNext := cSTA_EXTENDBusy;
		END_IF
	END_IF




//--------------------------------------------------------------------------------------
// Exit action
	IF (me.StateMachine.intState<>me.StateMachine.intStateNext) THEN
		SIf.Cur.udiMoveTimeRetract := me.StateMachine.udiTimeInState_ms;
	END_IF
END_METHOD

METHOD getCtrlSIf : POINTER TO T_Ctrl_SIf_CYL
getCtrlSIf := ADR(SIf);
END_METHOD

METHOD PROTECTED sta_PON : BOOL
// state implemetation
//--------------------------------------------------------------------------------------
// Entry action
	IF (me.StateMachine.intState<>me.StateMachine.intStateLastCycle) THEN
		me.StateMachine.intStateLastCycle := me.StateMachine.intState;
		
	END_IF


//--------------------------------------------------------------------------------------
// Cyclic action
	IF (me.StateMachine.intState=me.StateMachine.intStateLastCycle) THEN
		
		;
		
		
		// State Change Condition
		IF(me.intCmd=cCMD_OFF) THEN
			me.StateMachine.intStateNext := cSTA_OFFBusy;
		ELSIF(me.intCmd=cCMD_STOP) THEN
			me.StateMachine.intStateNext := cSTA_STOPBusy;
		ELSIF(me.intCmd=cCMD_RETRACT) THEN
			me.StateMachine.intStateNext := cSTA_RETRACTBusy;
		ELSIF (me.intCmd=cCMD_EXTEND) THEN
			me.StateMachine.intStateNext := cSTA_EXTENDBusy;
		END_IF
	END_IF




//--------------------------------------------------------------------------------------
// Exit action
	IF (me.StateMachine.intState<>me.StateMachine.intStateNext) THEN
		;
	END_IF
END_METHOD

METHOD PROTECTED CtrlInit : BOOL
SUPER^.CtrlInit();
END_METHOD

METHOD PROTECTED getCmdState : STRING
VAR_INPUT
	intCmdState: INT;
	bolState: BOOL;
END_VAR
getCmdState := SUPER^.getCmdState(intCmdState:=intCmdState,bolState:=bolState); // get global/base defined cmds/states
IF (getCmdState='') THEN // global not defined get local
	// get string cmd/state string information in runtime
	IF (bolState=FALSE) THEN
		// cmd's
		CASE intCmdState OF
			cCMD_RETRACT: 
				getCmdState := 'cCMD_RETRACT';
			cCMD_EXTEND: 
				getCmdState := 'cCMD_EXTEND';
		END_CASE;
	ELSE
	
	// cmd's
		CASE intCmdState OF
			cSTA_RETRACTBusy: 
				getCmdState := 'cSTA_RETRACTBusy';
			cSTA_RETRACT: 
				getCmdState := 'cSTA_RETRACT';
			cSTA_EXTENDBusy: 
				getCmdState := 'cSTA_EXTENDBusy';
			cCMD_EXTEND: 
				getCmdState := 'cCMD_EXTEND';
		END_CASE;
	END_IF
END_IF
END_METHOD

METHOD PROTECTED sta_OFF : BOOL
// state implemetation
//--------------------------------------------------------------------------------------
// Entry action
	IF (me.StateMachine.intState<>me.StateMachine.intStateLastCycle) THEN
		me.StateMachine.intStateLastCycle := me.StateMachine.intState;
		
	END_IF


//--------------------------------------------------------------------------------------
// Cyclic action
	IF (me.StateMachine.intState=me.StateMachine.intStateLastCycle) THEN
		
		;
		
		
		// State Change Condition
		IF (me.intCmd=cCMD_STOP) THEN
			// sensor retract always on cylinder
			me.StateMachine.intStateNext :=  cSTA_STOPBusy;
		ELSIF (me.intCmd=cCMD_EXTEND) THEN 
			me.StateMachine.intStateNext := cSTA_EXTENDBusy;
		ELSIF(me.intCmd=cCMD_RETRACT) THEN
			me.StateMachine.intStateNext := cSTA_RETRACTBusy;
		END_IF
	END_IF




//--------------------------------------------------------------------------------------
// Exit action
	IF (me.StateMachine.intState<>me.StateMachine.intStateNext) THEN
		;
	END_IF
END_METHOD

METHOD PROTECTED sta_OFFBusy : BOOL
// state implemetation
//--------------------------------------------------------------------------------------
// Entry action
	IF (me.StateMachine.intState<>me.StateMachine.intStateLastCycle) THEN
		me.StateMachine.intStateLastCycle := me.StateMachine.intState;
		
	END_IF


//--------------------------------------------------------------------------------------
// Cyclic action
	IF (me.StateMachine.intState=me.StateMachine.intStateLastCycle) THEN
		
		// switch off?
		IF (SIf.Cfg.eTyp = E_Typ_CYL.Valve1_Sensor0) OR (SIf.Cfg.eTyp = E_Typ_CYL.Valve1_Sensor2) 
			OR (SIf.Cfg.eTyp = E_Typ_CYL.Valve1_SensorExtended) OR (SIf.Cfg.eTyp = E_Typ_CYL.Valve1_SensorRetracted) THEN
			// monostabil valve -> do nothing
			;
		ELSE
			// bistable valve -> switch both off
			SIf.Out.bolExtend.intern := FALSE;
			SIf.Out.bolRetract.intern := FALSE;
		END_IF
		
		
		
		// State Change Condition
		IF (FALSE) THEN
			;
		ELSIF (TRUE) THEN
			me.StateMachine.intStateNext := cSTA_OFF;
		END_IF
	END_IF




//--------------------------------------------------------------------------------------
// Exit action
	IF (me.StateMachine.intState<>me.StateMachine.intStateNext) THEN
		;
	END_IF
END_METHOD

METHOD PROTECTED sta_STOP : BOOL
// state implemetation
//--------------------------------------------------------------------------------------
// Entry action
	IF (me.StateMachine.intState<>me.StateMachine.intStateLastCycle) THEN
		me.StateMachine.intStateLastCycle := me.StateMachine.intState;
		
	END_IF


//--------------------------------------------------------------------------------------
// Cyclic action
	IF (me.StateMachine.intState=me.StateMachine.intStateLastCycle) THEN
		
		;
		
		
		// State Change Condition
		IF (me.intCmd=cCMD_OFF) THEN
			// sensor retract always on cylinder
			me.StateMachine.intStateNext :=  cSTA_OFFBusy;
		ELSIF (me.intCmd=cCMD_EXTEND) THEN 
			me.StateMachine.intStateNext := cSTA_EXTENDBusy;
		ELSIF(me.intCmd=cCMD_RETRACT) THEN
			me.StateMachine.intStateNext := cSTA_RETRACTBusy;
		END_IF
	END_IF




//--------------------------------------------------------------------------------------
// Exit action
	IF (me.StateMachine.intState<>me.StateMachine.intStateNext) THEN
		;
	END_IF
END_METHOD

METHOD PROTECTED sta_STOPBusy : BOOL
// state implemetation
//--------------------------------------------------------------------------------------
// Entry action
	IF (me.StateMachine.intState<>me.StateMachine.intStateLastCycle) THEN
		me.StateMachine.intStateLastCycle := me.StateMachine.intState;
		
	END_IF


//--------------------------------------------------------------------------------------
// Cyclic action
	IF (me.StateMachine.intState=me.StateMachine.intStateLastCycle) THEN
		
		// switch off?
		IF (SIf.Cfg.eTyp = E_Typ_CYL.Valve1_Sensor0) OR (SIf.Cfg.eTyp = E_Typ_CYL.Valve1_Sensor2) 
			OR (SIf.Cfg.eTyp = E_Typ_CYL.Valve1_SensorExtended) OR (SIf.Cfg.eTyp = E_Typ_CYL.Valve1_SensorRetracted) THEN
			// monostabil valve -> do nothing
			;
		ELSE
			// bistable valve -> switch both on -> block at position
			SIf.Out.bolExtend.intern := TRUE;
			SIf.Out.bolRetract.intern := TRUE;
		END_IF
		
		
		
		// State Change Condition
		IF (FALSE) THEN
			;
		ELSIF (TRUE) THEN
			me.StateMachine.intStateNext := cSTA_STOP;
		END_IF
	END_IF




//--------------------------------------------------------------------------------------
// Exit action
	IF (me.StateMachine.intState<>me.StateMachine.intStateNext) THEN
		;
	END_IF
END_METHOD

END_FUNCTION_BLOCK

// ---- POUs/BaseCtrl/FB_CtrlBase.TcPOU
{attribute 'reflection' := ''}
FUNCTION_BLOCK FB_CtrlBase IMPLEMENTS I_CtrlBase
VAR
	///Commen interface struct for public access
	CIf: T_Ctrl_CIf;
	///basic local controller class struct
	me: T_Ctrl_Class;
	fbSimulationTimer: TON;
	{attribute 'instance-path' := ''}
	{attribute 'noinit' := ''}
	strMyInstancePath: STRING;
END_VAR

(*__________________________________________________________________________________________________
¦	
¦	Vistaprint Schweiz GmbH
¦	CH - 8401 Winterthur
¦
¦	www.vistaprint.ch - info@vistaprint.ch
¦___________________________________________________________________________________________________

Function desription:
Basic controller implementation. This Controller should be the base father controller for all in the
feature implemented ctontroller classes.


History:
Version		Date			Author		Comment
---------------------------------------------------------------------------------------------------
0.00.1		25.04.2013		AVME/KVO	Start history


___________________________________________________________________________________________________*)


IF (me.bolActivate) THEN // cyclic call enabled
	
	IF (CIf.Info.bolInitDone=FALSE) THEN // first cycle -> init
		CtrlInit();
		CIf.Info.bolInitDone := TRUE;
	ELSE
		CycleStartDuty();
	
		Always();
		
		StateMachine();
		
		CycleEndDuty();
	END_IF
	
END_IF;

METHOD iniCtrlArray : BOOL
VAR_INPUT
	p_pCtrlArray: POINTER TO POINTER TO FB_CtrlBase;
	intCtrlID: INT;
END_VAR
iniCtrlArray := FALSE;

IF (TRUE) THEN//e_CtrlID <= E_CtrlId.E_CtrlIdMax) THEN
	p_pCtrlArray[intCtrlID] := THIS;
	THIS^.CIf.Info.intCtrlID := intCtrlID;
	iniCtrlArray := TRUE;
END_IF
END_METHOD

METHOD FB_init : BOOL
VAR_INPUT
	///if TRUE, the retain variables are initialized (warm start / cold start)
	bInitRetains: BOOL;
	///if TRUE, the instance afterwards gets moved into the copy code (online change)
	bInCopyCode: BOOL;
END_VAR
//------------------------------------------------------------------------------------------------------------------------
// enable cyclic call
me.bolActivate := TRUE;
// reset init flag
CIf.Info.bolInitDone := FALSE;

//------------------------------------------------------------------------------------------------------------------------
// to manually change in new FUB implementation!!!
// define valid commands for this controller
CIf.Job.aCmdList[0].intCmd := cCMD_PON;
CIf.Job.aCmdList[0].strName := 'Power On';
CIf.Job.aCmdList[0].bolAvailable := TRUE;

CIf.Job.aCmdList[1].intCmd := cCMD_OFF; // for test simulation single answer
CIf.Job.aCmdList[1].strName := 'Off';
CIf.Job.aCmdList[1].bolAvailable := TRUE;

// set name of class/typ
CIf.Info.strType := 'FB_CtrlBase'; 

// for tests
CIf.SwCfg.bolExist := TRUE;
CIf.SwCfg.bolSimulation := TRUE;

//------------------------------------------------------------------------------------------------------------------------
CIf.Info.strName := getStrInstanceName(strMyInstancePath); // get name of instance
END_METHOD

METHOD PROTECTED StateMachine : BOOL

// main statemachine of base controller
CASE me.StateMachine.intState OF
    cSTA_PONBusy: 
        THIS^.sta_PONBusy();
    cSTA_PON: 
        THIS^.sta_PON();
	cSTA_OFFBusy: 
        THIS^.sta_OFFBusy();
    cSTA_OFF: 
        THIS^.sta_OFF();
    cSTA_ERROR: 
        THIS^.sta_ERROR();
    cSTA_ERRORQuit: 
        THIS^.sta_ERRORQuit();
    cSTA_SINGLE_ANSWER: 
        THIS^.sta_SINGLE_ANSWER();
END_CASE;
END_METHOD

METHOD PROTECTED sta_PONBusy : BOOL
// state implemetation
//--------------------------------------------------------------------------------------
// Entry action
	IF (me.StateMachine.intState<>me.StateMachine.intStateLastCycle) THEN
		me.StateMachine.intStateLastCycle := me.StateMachine.intState;
		
	END_IF


//--------------------------------------------------------------------------------------
// Cyclic action
	IF (me.StateMachine.intState=me.StateMachine.intStateLastCycle) THEN
		
		;
		
		
		// State Change Condition
		IF (FALSE) THEN
			;
		ELSIF (TRUE) THEN
			me.StateMachine.intStateNext := cSTA_PON;
		END_IF
	END_IF




//--------------------------------------------------------------------------------------
// Exit action
	IF (me.StateMachine.intState<>me.StateMachine.intStateNext) THEN
		;
	END_IF
END_METHOD

METHOD PROTECTED sta_PON : BOOL
// state implemetation
//--------------------------------------------------------------------------------------
// Entry action
	IF (me.StateMachine.intState<>me.StateMachine.intStateLastCycle) THEN
		me.StateMachine.intStateLastCycle := me.StateMachine.intState;
		
	END_IF


//--------------------------------------------------------------------------------------
// Cyclic action
	IF (me.StateMachine.intState=me.StateMachine.intStateLastCycle) THEN
		
		;
		
		
		// State Change Condition
		IF (FALSE) THEN
			;
		ELSIF (me.intCmd=cCMD_OFF) THEN
			me.StateMachine.intStateNext := cSTA_OFFBusy;
		END_IF
	END_IF




//--------------------------------------------------------------------------------------
// Exit action
	IF (me.StateMachine.intState<>me.StateMachine.intStateNext) THEN
		;
	END_IF
END_METHOD

METHOD PROTECTED sta_ERROR : BOOL
// state implemetation
//--------------------------------------------------------------------------------------
// Entry action
	IF (me.StateMachine.intState<>me.StateMachine.intStateHistory) THEN
		me.StateMachine.intStateHistory := me.StateMachine.intStateLastCycle; // -> possibillity to go back to state before error
		me.StateMachine.intStateLastCycle := me.StateMachine.intState;
		
	END_IF


//--------------------------------------------------------------------------------------
// Cyclic action
	IF (me.StateMachine.intState=me.StateMachine.intStateLastCycle) THEN
		
		;
		
		
		// State Change Condition
		IF (CIf.Job.bolAlmReset = TRUE) THEN
			me.StateMachine.intStateNext := cSTA_ERRORQuit;
		END_IF
	END_IF




//--------------------------------------------------------------------------------------
// Exit action
	IF (me.StateMachine.intState<>me.StateMachine.intStateNext) THEN
		;
	END_IF
END_METHOD

METHOD PROTECTED sta_ERRORQuit : BOOL
// state implemetation
//--------------------------------------------------------------------------------------
// Entry action
	IF (me.StateMachine.intState<>me.StateMachine.intStateLastCycle) THEN
		me.StateMachine.intStateLastCycle := me.StateMachine.intState;
		
	END_IF


//--------------------------------------------------------------------------------------
// Cyclic action
	IF (me.StateMachine.intState=me.StateMachine.intStateLastCycle) THEN
		
		;
		// evtl. wait time if reset of device is necessary and then decide to go to states or ERROR state
		IF (CIf.Job.bolAlmReset = TRUE) THEN
			CIf.Job.eMe_ActivAlmClass := E_AlmClass.NONE; // reset feedback channel for parent
			CIf.Job.bolAlmReset := FALSE;
		END_IF
		
		// State Change Condition
		IF (CIf.Job.bolAlmReset = FALSE) OR (me.StateMachine.intStateHistory<=cSTA_PON) THEN
			me.StateMachine.intStateNext := cSTA_PONBusy;
		END_IF
	END_IF




//--------------------------------------------------------------------------------------
// Exit action
	IF (me.StateMachine.intState<>me.StateMachine.intStateNext) THEN
		;
	END_IF
END_METHOD

METHOD PROTECTED sta_SINGLE_ANSWER : BOOL
// state implemetation of SINGLE_ANSWER
//--------------------------------------------------------------------------------------
// Entry action
	IF (me.StateMachine.intState<>me.StateMachine.intStateLastCycle) THEN
		me.StateMachine.intStateLastCycle := me.StateMachine.intState;
		
	END_IF


//--------------------------------------------------------------------------------------
// Cyclic action
	IF (me.StateMachine.intState=me.StateMachine.intStateLastCycle) THEN
		
		IF ((me.intCmd<>cCMD_INITIALIZED) AND (me.intCmd<>cCMD_DONE)) THEN
			IF (THIS^.CheckCmdValid()=TRUE) THEN
				IF (me.intCmd<>me.intCmdLast) THEN
					me.StateMachine.udiTimeInState_ms := 0;  // reset timer
				END_IF
				IF (me.StateMachine.udiTimeInState_ms >= me.StateMachine.udiStateSimSetTime_ms) THEN
					CIf.Job.intState := me.intCmd; // simulate final state
				ELSE
					CIf.Job.intState := me.intCmd-1; // simulate busy state
				END_IF
			END_IF
		END_IF
		
		// State Change Condition
		IF (FALSE) THEN
			;
		ELSIF (CIf.SwCfg.bolExist=TRUE) THEN
			me.StateMachine.intStateNext := cSTA_PONBusy;
		END_IF
	END_IF




//--------------------------------------------------------------------------------------
// Exit action
	IF (me.StateMachine.intState<>me.StateMachine.intStateNext) THEN
		;
	END_IF
END_METHOD

METHOD PROTECTED CycleStartDuty : BOOL

	// --------------------------------------------------------------------------
	// input bridge
	// --------------------------------------------------------------------------
	THIS^.IoInBridge(); // digitale and analoge inputs read from hardware or forcing

	// --------------------------------------------------------------------------
	// check alarm recation class of master													
	// --------------------------------------------------------------------------
	THIS^.CheckParentAlmClass();
	
	// ----------------------------------------------------------------------------------
	// check the highest active alarm -> set local class
	// ----------------------------------------------------------------------------------
	IF (me.Alarm.eParent_ActivAlmClass>CIf.job.eMe_ActivAlmClass) THEN
		me.Alarm.eActivAlmClass := me.Alarm.eParent_ActivAlmClass;
	ELSE
		me.Alarm.eActivAlmClass := CIf.job.eMe_ActivAlmClass;
	END_IF
	
	// --------------------------------------------------------------------------
	// get command											
	// --------------------------------------------------------------------------
	IF (CIf.Job.eMode = E_Mode.MANU) THEN
		me.intCmd := CIf.Job.intMCmd;  
	ELSE
		IF (me.eModeHistory <> E_MODE.AUTO) THEN
			CIf.Job.intMCmd:= cCMD_DONE;	// reset manual command
			me.bolChangeBackToAUTO := TRUE;	// switch off  or .....
		END_IF
		CIf.Job.eMode := E_MODE.AUTO;
		me.intCmd := CIf.Job.intACmd;
	END_IF
	CIf.Job.strCmd := THIS^.getCmdState(intCmdState:=me.intCmd,bolState:=FALSE);
END_METHOD

METHOD PROTECTED CycleEndDuty : BOOL

me.eModeHistory := CIf.Job.eMode;				// save mode to detect mode switches
me.intCmdLast := me.intCmd;
IF (me.StateMachine.intState<>cSTA_SINGLE_ANSWER) THEN // only if no simulation is active
	CIf.Job.intState := me.StateMachine.intState;		// set information of actual state to controller interface
	CIf.Job.strState := THIS^.getCmdState(intCmdState:=CIf.Job.intState,bolState:=TRUE);
ELSE
	CIf.Job.strState :=  TC2_STANDARD.CONCAT(STR1:='SINGLE_ANSWER-',STR2:=THIS^.getCmdState(intCmdState:=CIf.Job.intState,bolState:=TRUE));
END_IF

	
IF (me.StateMachine.intState<>me.StateMachine.intStateNext) THEN
	me.StateMachine.intState := me.StateMachine.intStateNext;  // set next state for next cycle
	me.StateMachine.udiTimeInState_ms := 0; // reset timer
	// log state change -> open point
ELSE
	// increment time in state	
	me.StateMachine.udiTimeInState_ms := me.StateMachine.udiTimeInState_ms + me.FUBInfo.udiSample_ms;
END_IF

// --------------------------------------------------------------------------
// Final state reached -> reset command
// --------------------------------------------------------------------------
IF (CIf.Job.intState=me.intCmd) THEN 
	CIf.Job.intACmd := cCMD_DONE;
	CIf.Job.intMCmd := cCMD_DONE;
END_IF

// --------------------------------------------------------------------------
// reset local alarm class
// --------------------------------------------------------------------------
IF (CIf.Job.bolAlmReset=TRUE) AND (CIf.Job.intState<>cSTA_ERROR) AND (CIf.Job.intState<>cSTA_ERRORQuit) THEN
	CIf.Job.eMe_ActivAlmClass := E_AlmClass.NONE;
	CIf.Job.bolAlmReset := FALSE;
END_IF

// --------------------------------------------------------------------------
// output bridge
// --------------------------------------------------------------------------
THIS^.IoOutBridge();	// digitale and analoge outputs or forcing write to hardware
END_METHOD

METHOD PROTECTED IoInBridge : BOOL
// digitale and analoge inputs read from hardware or forcing
IF (CIf.SwCfg.bolSimulation = FALSE) THEN
	//KVO??? alternative only without feedback getIn(ctrl.ifc.Job.bol_Force ,ADR(ctrl.In.bol_PosSwitchBasicDefTyp);
	//ctrl.In.bol_PosSwitchBasicDefTyp.intern := getIn(ctrl.ifc.Job.bol_Force ,ADR(ctrl.In.bol_PosSwitchBasicDefTyp);
ELSE
	//simulation of global IO
END_IF
END_METHOD

METHOD PRIVATE CheckParentAlmClass : BOOL
// --------------------------------------------------------------------------
// check alarm recation class of master													
// --------------------------------------------------------------------------
IF (CIf.Job.eParent_ActivAlmClass = E_AlmClass.EOFF) THEN
	me.Alarm.eParent_ActivAlmClass := E_AlmClass.EOFF;
	// prevent automatic restart in manual or automatic
	CIf.job.intACmd := cCMD_DONE;
	CIf.job.intMCmd  := cCMD_DONE;
ELSE
	me.Alarm.eParent_ActivAlmClass := E_AlmClass.NONE;
END_IF
END_METHOD

METHOD PROTECTED Always : BOOL
// ----------------------------------------------------------------------------------
// cyclic actions outside of statemachine
IF (me.StateMachine.intState<>cSTA_SINGLE_ANSWER) THEN
	
	; // always error supervision
	
END_IF

// ----------------------------------------------------------------------------------
// Conditions Always
IF (me.bolChangeBackToAUTO=TRUE) THEN // switch mode to automatic switch off controller
	me.StateMachine.intStateNext := cSTA_OFFBusy;
	me.bolChangeBackToAUTO := FALSE;
END_IF

IF ((me.StateMachine.intState=cSTA_INITIALIZED) OR (me.intCmd=cCMD_PON)) AND (me.StateMachine.intState<>cSTA_PONBusy)  AND (me.StateMachine.intState<>cSTA_PON) THEN // switch after startup to PONBusy
	me.StateMachine.intStateNext := cSTA_PONBusy;
END_IF

IF (CIf.SwCfg.bolExist=FALSE) AND (me.StateMachine.intState<>cSTA_SINGLE_ANSWER) THEN // hardware of controller does not exist
	me.StateMachine.intStateNext := cSTA_SINGLE_ANSWER;
END_IF
END_METHOD

METHOD PRIVATE CheckCmdValid : BOOL
VAR
	ii: UINT;
END_VAR
CheckCmdValid := FALSE;
FOR ii:=0 TO cMaxCmdPerCtrl BY 1 DO
	// check if a valid cmd
	IF (CIf.Job.aCmdList[ii].intCmd=cCMD_INITIALIZED) OR (CIf.Job.aCmdList[ii].intCmd=cCMD_DONE) THEN
		EXIT; // end for
	END_IF
	// check if a in this ctrl implemented cmd
	IF (CIf.Job.aCmdList[ii].intCmd=me.intCmd) THEN
		CheckCmdValid := TRUE;
	END_IF
END_FOR
END_METHOD

METHOD PROTECTED IoOutBridge : BOOL
// digitale and analoge inputs read from hardware or forcing
IF (CIf.SwCfg.bolSimulation = FALSE) THEN


//KVO??? alternative only without feedback getIn(ctrl.ifc.Job.bol_Force ,ADR(ctrl.In.bol_PosSwitchBasicDefTyp);
	// check interlocks to prevent damages
	//IF (SIf.Ilk.bolOverwrite=FALSE) THEN
		//IF (SIf.Ilk.bolOut=FALSE) THEN
			//ctrl.Out.bolOut.map := setOut(ctrl.ifc.Job.bol_Force ,ADR(ctrl.Out.bolOut);
		//ELSE
			// switch off???
			// error??
		//END_IF
	//end_if


END_IF
END_METHOD

METHOD getCtrlCIf : POINTER TO T_Ctrl_CIf
getCtrlCIf := adr(THIS^.CIf);
END_METHOD

METHOD PROTECTED CtrlInit : BOOL
VAR
	udiTaskCnt: UDINT;
	fbGETCURTASKINDEX: Tc2_System.GETCURTASKINDEX;
END_VAR

//automatic read out infos about FUB
udiTaskCnt := TwinCAT_SystemInfoVarList._AppInfo.TaskCnt;
fbGETCURTASKINDEX();
udiTaskCnt := fbGETCURTASKINDEX.index;
me.FUBInfo.udiSample_ms := TwinCAT_SystemInfoVarList._TaskInfo[UDINT_TO_DINT(udiTaskCnt)].CycleTime/10000; //[ms] X[100ns]/10000 -> [ms]
END_METHOD

METHOD PROTECTED getCmdState : STRING
VAR_INPUT
	intCmdState: INT;
	bolState: BOOL;
END_VAR
// get string cmd/state string information in runtime
IF (bolState=FALSE) THEN
	// cmd's
	CASE intCmdState OF
		cCMD_DONE: 
			getCmdState := 'cCMD_DONE';
		cCMD_INITIALIZED: 
			getCmdState := 'cCMD_INITIALIZED';
		cCMD_PON: 
			getCmdState := 'cCMD_PON';
		cCMD_EOFF: 
			getCmdState := 'cCMD_EOFF';
		cCMD_OFF: 
			getCmdState := 'cCMD_OFF';
		cCMD_INIT: 
			getCmdState := 'cCMD_INIT';
		cCMD_RUN: 
			getCmdState := 'cCMD_RUN';
		cCMD_STOP: 
			getCmdState := 'cCMD_STOP';
		cCMD_TSTOP: 
			getCmdState := 'cCMD_TSTOP';
	END_CASE;
ELSE

// cmd's
	CASE intCmdState OF
		cSTA_DONE: 
			getCmdState := 'cSTA_DONE';
		cSTA_INITIALIZED: 
			getCmdState := 'cSTA_INITIALIZED';
		cSTA_PONBusy: 
			getCmdState := 'cSTA_PONBusy';
		cSTA_PON: 
			getCmdState := 'cSTA_PON';
		cSTA_EOFFBusy: 
			getCmdState := 'cSTA_EOFFBusy';
		cSTA_EOFF: 
			getCmdState := 'cSTA_EOFF';
		cSTA_OFFBusy: 
			getCmdState := 'cSTA_OFFBusy';
		cSTA_OFF: 
			getCmdState := 'cSTA_OFF';
		cSTA_INITBusy: 
			getCmdState := 'cSTA_INITBusy';
		cSTA_INIT: 
			getCmdState := 'cSTA_INIT';
		cSTA_RUNBusy: 
			getCmdState := 'cSTA_RUNBusy';
		cSTA_RUN: 
			getCmdState := 'cSTA_RUN';
		cSTA_STOPBusy: 
			getCmdState := 'cSTA_STOPBusy';
		cSTA_STOP: 
			getCmdState := 'cSTA_STOP';
		cSTA_TSTOPBusy: 
			getCmdState := 'cSTA_TSTOPBusy';
		cSTA_TSTOP: 
			getCmdState := 'cSTA_TSTOP';
			
		cSTA_ERROR: 
			getCmdState := 'cSTA_ERROR';
		cSTA_ERRORQuit: 
			getCmdState := 'cSTA_ERRORQuit';
		cSTA_SINGLE_ANSWER: 
			getCmdState := 'cSTA_SINGLE_ANSWER';
	END_CASE;
END_IF
END_METHOD

METHOD PROTECTED sta_OFF : BOOL
// state implemetation
//--------------------------------------------------------------------------------------
// Entry action
	IF (me.StateMachine.intState<>me.StateMachine.intStateLastCycle) THEN
		me.StateMachine.intStateLastCycle := me.StateMachine.intState;
		
	END_IF


//--------------------------------------------------------------------------------------
// Cyclic action
	IF (me.StateMachine.intState=me.StateMachine.intStateLastCycle) THEN
		
		;
		
		
		// State Change Condition
		IF (FALSE) THEN
			;
		ELSIF (TRUE) THEN
			;	//me.StateMachine.intStateNext := cSTA_PON;
		END_IF
	END_IF




//--------------------------------------------------------------------------------------
// Exit action
	IF (me.StateMachine.intState<>me.StateMachine.intStateNext) THEN
		;
	END_IF
END_METHOD

METHOD PROTECTED sta_OFFBusy : BOOL
// state implemetation
//--------------------------------------------------------------------------------------
// Entry action
	IF (me.StateMachine.intState<>me.StateMachine.intStateLastCycle) THEN
		me.StateMachine.intStateLastCycle := me.StateMachine.intState;
		
	END_IF


//--------------------------------------------------------------------------------------
// Cyclic action
	IF (me.StateMachine.intState=me.StateMachine.intStateLastCycle) THEN
		
		;
		
		
		// State Change Condition
		IF (FALSE) THEN
			;
		ELSIF (TRUE) THEN
			me.StateMachine.intStateNext := cSTA_OFF;
		END_IF
	END_IF




//--------------------------------------------------------------------------------------
// Exit action
	IF (me.StateMachine.intState<>me.StateMachine.intStateNext) THEN
		;
	END_IF
END_METHOD

END_FUNCTION_BLOCK

// ---- POUs/Utility Functions/getStrInstanceName.TcPOU
FUNCTION getStrInstanceName : T_MaxString
VAR_INPUT
	///'C:\TwinCAT\Plc\Project01\Data.txt';
	strPathName: T_MaxString;
END_VAR
VAR
	strDrive: STRING(3);
	strDir: T_MaxString;
	strFileName: T_MaxString;
	strExt: T_MaxString;
	bolSuccess: BOOL;
END_VAR


bolSuccess := F_SplitPathName( sPathName := strPathName,
                                sDrive := strDrive,
                                sDir := strDir,
                                sFileName := strFileName,
                                sExt := strExt );
								
								getStrInstanceName := MID (strExt,TC2_STANDARD.LEN(strExt),2);

END_FUNCTION

// ---- POUs/Utility Functions/getInBol.TcPOU
FUNCTION getInBol : BOOL
VAR_INPUT
	bol_GlobalEnableForce: BOOL;
	p_Input: POINTER TO T_Ctrl_IoBool;
END_VAR

p_Input^.state := p_Input^.map;

IF (p_Input^.EnForce OR bol_GlobalEnableForce) THEN
	p_Input^.intern := p_Input^.force;
ELSE
	p_Input^.intern := p_Input^.map;
END_IF;

getInBol := p_Input^.intern;

END_FUNCTION

// ---- POUs/Utility Functions/setOutBol.TcPOU
FUNCTION setOutBol : BOOL
VAR_INPUT
	bol_GlobalEnableForce: BOOL;
	p_Output: POINTER TO T_Ctrl_IoBool;
END_VAR

// Copy real values
p_Output^.state := p_Output^.intern;

IF (p_Output^.EnForce OR bol_GlobalEnableForce) THEN
	p_Output^.map := p_Output^.force;
ELSE
	p_Output^.map := p_Output^.intern;
END_IF;

setOutBol := p_Output^.map;

END_FUNCTION

// ---- POUs/Controller/Lvl2/MOD/FB_MOD.TcPOU
FUNCTION_BLOCK FB_MOD EXTENDS FB_CtrlBase
VAR_INPUT
	///pointer to function block
	p_fbHOR: POINTER TO FB_CYL;
	///pointer to function block
	p_fbVER: POINTER TO FB_CYL;
END_VAR
VAR
	///Specific interface struct for public access
	SIf: T_Ctrl_SIf_MOD;
	pHOR_CIF: POINTER TO T_Ctrl_CIf;
	pVER_CIF: POINTER TO T_Ctrl_CIf;
	stSubSate: T_MOD_RUN_StateMachine;
	bolfpCmd: BOOL;
	bolfpInit: BOOL;
END_VAR

(*__________________________________________________________________________________________________
¦	
¦	Vistaprint Schweiz GmbH
¦	CH - 8401 Winterthur
¦
¦	www.vistaprint.ch - info@vistaprint.ch
¦___________________________________________________________________________________________________

Function desription:
This controller is an example of a level 2 modul controller. It has two cylinder FUB as childs. 
One is for up and down and the other is for a movement horizontal.(pick and place)


History:
Version		Date			Author		Comment
---------------------------------------------------------------------------------------------------
0.00.1		02.05.2013		AVME/KVO	Start history


___________________________________________________________________________________________________*)

// check if child pointer valid
IF (me.bolActivate) AND (p_fbHOR<>0) AND (p_fbVER<>0) THEN // cyclic call enabled
	
	IF (CIf.Info.bolInitDone=FALSE) THEN // first cycle -> init
		CtrlInit();
		CIf.Info.bolInitDone := TRUE;
	ELSE
		CycleStartDuty();
	
		Always();
		
		StateMachine();
		THIS^.CIf.Job.strSubState := stSubSate.strState; // entry substate info to common interface
		
		CycleEndDuty();
	END_IF
	
END_IF;

METHOD FB_init : BOOL
VAR_INPUT
	///if TRUE, the retain variables are initialized (warm start / cold start)
	bInitRetains: BOOL;
	///if TRUE, the instance afterwards gets moved into the copy code (online change)
	bInCopyCode: BOOL;
END_VAR
VAR
	ii: UINT;
END_VAR
//------------------------------------------------------------------------------------------------------------------------
// to manually change in new FUB implementation!!!
// define valid commands for this controller
FOR ii:= 0 TO (SIZEOF(CIf.Job.aCmdList)/SIZEOF(CIf.Job.aCmdList[0])-1) BY 1 DO
	IF (CIf.Job.aCmdList[ii].intCmd=cSTA_INITIALIZED) THEN
		// found first empty array element
		EXIT;
	END_IF
END_FOR

CIf.Job.aCmdList[ii].intCmd := cSTA_INIT;
CIf.Job.aCmdList[ii].strName := 'Init';
CIf.Job.aCmdList[ii].bolAvailable := TRUE;
ii := ii +1;
CIf.Job.aCmdList[ii].intCmd := cSTA_RUN;
CIf.Job.aCmdList[ii].strName := 'Run';
CIf.Job.aCmdList[ii].bolAvailable := TRUE;

// set name of class/typ
CIf.Info.strType := 'FB_MOD'; 

// set alarm class
SIf.Alm[1].eAlmClass := E_AlmClass.EOFF;
SIf.Alm[2].eAlmClass := E_AlmClass.OFF;
SIf.Alm[3].eAlmClass := E_AlmClass.STOP;
SIf.Alm[4].eAlmClass := E_AlmClass.TSTOP;
SIf.Alm[5].eAlmClass := E_AlmClass.INFO;
SIf.Alm[6].eAlmClass := E_AlmClass.WARNING;

// for tests
CIf.SwCfg.bolSimulation := FALSE;
SIf.Par.udiWaitPick_ms := 15000;
END_METHOD

METHOD PROTECTED StateMachine : BOOL
SUPER^.StateMachine();

// main statemachine of base controller
CASE me.StateMachine.intState OF
	 cSTA_OFFBusy: 
        THIS^.sta_OFFBusy();
    cSTA_OFF: 
        THIS^.sta_OFF();
    cSTA_INITBusy: 
        THIS^.sta_INITBusy();
    cSTA_INIT: 
        THIS^.sta_INIT();
    cSTA_RUNBusy: 
        THIS^.sta_RUNBusy();
    cSTA_RUN: 
        THIS^.sta_RUN();
END_CASE;
END_METHOD

METHOD PROTECTED sta_ERROR : BOOL
// state implemetation
//--------------------------------------------------------------------------------------
// Entry action
	IF (me.StateMachine.intState<>me.StateMachine.intStateHistory) THEN
		me.StateMachine.intStateHistory := me.StateMachine.intStateLastCycle; // -> possibillity to go back to state before error
		me.StateMachine.intStateLastCycle := me.StateMachine.intState;
		
	END_IF


//--------------------------------------------------------------------------------------
// Cyclic action
	IF (me.StateMachine.intState=me.StateMachine.intStateLastCycle) THEN
		
		;
		
		
		// State Change Condition
		IF (CIf.Job.bolAlmReset = TRUE) THEN
			me.StateMachine.intStateNext := cSTA_ERRORQuit;
		END_IF
	END_IF




//--------------------------------------------------------------------------------------
// Exit action
	IF (me.StateMachine.intState<>me.StateMachine.intStateNext) THEN
		;
	END_IF
END_METHOD

METHOD PROTECTED sta_ERRORQuit : BOOL
// state implemetation
//--------------------------------------------------------------------------------------
// Entry action
	IF (me.StateMachine.intState<>me.StateMachine.intStateLastCycle) THEN
		me.StateMachine.intStateLastCycle := me.StateMachine.intState;
		
	END_IF


//--------------------------------------------------------------------------------------
// Cyclic action
	IF (me.StateMachine.intState=me.StateMachine.intStateLastCycle) THEN
		
		;
		// evtl. wait time if reset of device is necessary and then decide to go to states or ERROR state
		IF (CIf.Job.bolAlmReset = TRUE) THEN
			CIf.Job.eMe_ActivAlmClass := E_AlmClass.NONE; // reset feedback channel for parent
			CIf.Job.bolAlmReset := FALSE;
		END_IF
		
		// State Change Condition
		IF (CIf.Job.bolAlmReset = FALSE) THEN
			// State Change Condition
			IF ((CIf.Job.eParent_ActivAlmClass=E_AlmClass.EOFF) OR (CIf.Job.eParent_ActivAlmClass=E_AlmClass.OFF)) OR 
				((CIf.Job.eMe_ActivAlmClass=E_AlmClass.EOFF) OR (CIf.Job.eMe_ActivAlmClass=E_AlmClass.OFF)) THEN
				me.StateMachine.intStateNext := cSTA_OFFBusy;
			ELSIF (me.StateMachine.intStateHistory<=cSTA_PON) OR (me.intCmd=cSTA_PON) THEN
				me.StateMachine.intStateNext := cSTA_PONBusy;
			ELSIF(me.intCmd=cSTA_OFF) THEN
				me.StateMachine.intStateNext := cSTA_OFFBusy;
			ELSIF(me.intCmd=cSTA_INIT) THEN
				me.StateMachine.intStateNext := cSTA_INITBusy;
			ELSIF(me.intCmd=cSTA_RUN) THEN
				me.StateMachine.intStateNext := cSTA_INITBusy;
			END_IF
		END_IF
	END_IF




//--------------------------------------------------------------------------------------
// Exit action
	IF (me.StateMachine.intState<>me.StateMachine.intStateNext) THEN
		;
	END_IF
END_METHOD

METHOD PROTECTED sta_INITBusy : BOOL
// state implemetation
//--------------------------------------------------------------------------------------
// Entry action
	IF (me.StateMachine.intState<>me.StateMachine.intStateLastCycle) THEN
		me.StateMachine.intStateLastCycle := me.StateMachine.intState;
		
		
	END_IF


//--------------------------------------------------------------------------------------
// Cyclic action
	IF (me.StateMachine.intState=me.StateMachine.intStateLastCycle) THEN

		// Simulation
		IF (CIf.SwCfg.bolSimulation) THEN
			;
		END_IF
		
		// no change action
		IF (pVER_CIF^.Job.intState = cSTA_RETRACT) THEN
			pHOR_CIF^.Job.intACmd := cCMD_RETRACT; // go to home position of horizontal cylinder
		ELSE
			pVER_CIF^.Job.intACmd := cCMD_RETRACT; // cylinder move up, 
			// problem command could not set in entry because if VER in manual moved  during this step to extend....
		END_IF
		
		// State Change Condition
		IF ((me.Alarm.eActivAlmClass=E_AlmClass.EOFF) OR (me.Alarm.eActivAlmClass=E_AlmClass.OFF)) THEN
			me.StateMachine.intStateNext := cSTA_OFFBusy;
		ELSIF(me.intCmd=cSTA_OFF) THEN
			me.StateMachine.intStateNext := cSTA_OFFBusy;
		ELSIF (pVER_CIF^.Job.intState = cSTA_RETRACT) AND (pHOR_CIF^.Job.intState = cSTA_RETRACT) THEN
			me.StateMachine.intStateNext := cSTA_INIT;
		END_IF
	END_IF



//--------------------------------------------------------------------------------------
// Exit action
	IF (me.StateMachine.intState<>me.StateMachine.intStateNext) THEN
		;
	END_IF
END_METHOD

METHOD PROTECTED sta_INIT : BOOL
// state implemetation
//--------------------------------------------------------------------------------------
// Entry action
	IF (me.StateMachine.intState<>me.StateMachine.intStateLastCycle) THEN
		me.StateMachine.intStateLastCycle := me.StateMachine.intState;

	END_IF


//--------------------------------------------------------------------------------------
// Cyclic action
	IF (me.StateMachine.intState=me.StateMachine.intStateLastCycle) THEN

		// Simulation
		IF (CIf.SwCfg.bolSimulation) THEN
			;
		END_IF
		
		// State Change Condition
		// State Change Condition
		IF ((me.Alarm.eActivAlmClass=E_AlmClass.EOFF) OR (me.Alarm.eActivAlmClass=E_AlmClass.OFF)) THEN
			me.StateMachine.intStateNext := cSTA_OFFBusy;
		ELSIF(me.intCmd=cSTA_OFF) THEN
			me.StateMachine.intStateNext := cSTA_OFFBusy;
		ELSIF(me.intCmd=cSTA_RUN) THEN
			me.StateMachine.intStateNext := cSTA_RUNBusy;
		END_IF
	END_IF




//--------------------------------------------------------------------------------------
// Exit action
	IF (me.StateMachine.intState<>me.StateMachine.intStateNext) THEN
		;
	END_IF
END_METHOD

METHOD PROTECTED sta_OFF : BOOL
// state implemetation
//--------------------------------------------------------------------------------------
// Entry action
	IF (me.StateMachine.intState<>me.StateMachine.intStateLastCycle) THEN
		me.StateMachine.intStateLastCycle := me.StateMachine.intState;

	END_IF


//--------------------------------------------------------------------------------------
// Cyclic action
	IF (me.StateMachine.intState=me.StateMachine.intStateLastCycle) THEN

		// Simulation
		IF (CIf.SwCfg.bolSimulation) THEN
			;
		END_IF
		
		// State Change Condition
		IF ((me.Alarm.eActivAlmClass<>E_AlmClass.EOFF) AND (me.Alarm.eActivAlmClass<>E_AlmClass.OFF)) THEN
			// enable start - no important error active
			IF(me.intCmd=cSTA_INIT) THEN
				me.StateMachine.intStateNext := cSTA_INITBusy;
			ELSIF(me.intCmd=cSTA_RUN) THEN
				me.StateMachine.intStateNext := cSTA_INITBusy;
			END_IF
		END_IF
	END_IF




//--------------------------------------------------------------------------------------
// Exit action
	IF (me.StateMachine.intState<>me.StateMachine.intStateNext) THEN
		;
	END_IF
END_METHOD

METHOD PROTECTED sta_OFFBusy : BOOL
// state implemetation
//--------------------------------------------------------------------------------------
// Entry action
	IF (me.StateMachine.intState<>me.StateMachine.intStateLastCycle) THEN
		me.StateMachine.intStateLastCycle := me.StateMachine.intState;
		
		// no action needed
		
	END_IF


//--------------------------------------------------------------------------------------
// Cyclic action
	IF (me.StateMachine.intState=me.StateMachine.intStateLastCycle) THEN

		// Simulation
		IF (CIf.SwCfg.bolSimulation) THEN
			;
		END_IF
		
		// State Change Condition
		IF (TRUE) THEN
			me.StateMachine.intStateNext := cSTA_OFF;
		END_IF
	END_IF




//--------------------------------------------------------------------------------------
// Exit action
	IF (me.StateMachine.intState<>me.StateMachine.intStateNext) THEN
		;
	END_IF
END_METHOD

METHOD getCtrlSIf : POINTER TO T_Ctrl_SIf_CYL
getCtrlSIf := ADR(SIf);
END_METHOD

METHOD PROTECTED sta_PON : BOOL
// state implemetation
//--------------------------------------------------------------------------------------
// Entry action
	IF (me.StateMachine.intState<>me.StateMachine.intStateLastCycle) THEN
		me.StateMachine.intStateLastCycle := me.StateMachine.intState;
		
	END_IF


//--------------------------------------------------------------------------------------
// Cyclic action
	IF (me.StateMachine.intState=me.StateMachine.intStateLastCycle) THEN
		
		;
		
		
		// State Change Condition
		IF(me.intCmd=cSTA_OFF) OR (me.intCmd=cSTA_INIT) OR (me.intCmd=cSTA_RUN) THEN
			me.StateMachine.intStateNext := cSTA_OFFBusy;
		END_IF
	END_IF




//--------------------------------------------------------------------------------------
// Exit action
	IF (me.StateMachine.intState<>me.StateMachine.intStateNext) THEN
		;
	END_IF
END_METHOD

METHOD PROTECTED Always : BOOL
// ---------------------------------------------------------------------------------
// check child me and set parent alarm class
checkChildAlmClass();


// ----------------------------------------------------------------------------------
// cyclic actions outside of statemachine
IF (me.StateMachine.intState<>cSTA_SINGLE_ANSWER) THEN
	
	; // always error supervision
	
END_IF



// ----------------------------------------------------------------------------------
// Conditions Always
IF (me.bolChangeBackToAUTO=TRUE) THEN // switch mode to automatic switch off controller
	me.StateMachine.intStateNext := cSTA_OFFBusy;
	me.bolChangeBackToAUTO := FALSE;
END_IF

IF ((me.StateMachine.intState=cSTA_INITIALIZED) OR (me.intCmd=cCMD_PON)) THEN // switch after startup to PONBusy
	me.StateMachine.intStateNext := cSTA_PONBusy;
END_IF

IF (CIf.SwCfg.bolExist=FALSE) AND (me.StateMachine.intState<>cSTA_SINGLE_ANSWER) THEN // hardware of controller does not exist
	me.StateMachine.intStateNext := cSTA_SINGLE_ANSWER;
END_IF
END_METHOD

METHOD PROTECTED sta_PONBusy : BOOL
// state implemetation
//--------------------------------------------------------------------------------------
// Entry action
	IF (me.StateMachine.intState<>me.StateMachine.intStateLastCycle) THEN
		me.StateMachine.intStateLastCycle := me.StateMachine.intState;
		
	END_IF


//--------------------------------------------------------------------------------------
// Cyclic action
	IF (me.StateMachine.intState=me.StateMachine.intStateLastCycle) THEN
		
		pVER_CIF^.Job.intACmd := cCMD_PON;
		pHOR_CIF^.Job.intACmd := cCMD_PON;
		
		// State Change Condition
		IF (pVER_CIF^.Job.intState = cSTA_PON) AND (pHOR_CIF^.Job.intState = cSTA_PON) THEN
			me.StateMachine.intStateNext := cSTA_PON;
		ELSE
			;
			// timeout power on child not ok -> failure or log entry???
		END_IF
	END_IF




//--------------------------------------------------------------------------------------
// Exit action
	IF (me.StateMachine.intState<>me.StateMachine.intStateNext) THEN
		;
	END_IF
END_METHOD

METHOD PROTECTED sta_RUNBusy : BOOL
// state implemetation
//--------------------------------------------------------------------------------------
// Entry action
	IF (me.StateMachine.intState<>me.StateMachine.intStateLastCycle) THEN
		me.StateMachine.intStateLastCycle := me.StateMachine.intState;
		
		stSubSate.intState := cCMD_INITIALIZED; // init sub state machine
	END_IF


//--------------------------------------------------------------------------------------
// Cyclic action
	IF (me.StateMachine.intState=me.StateMachine.intStateLastCycle) THEN

		// Simulation
		IF (CIf.SwCfg.bolSimulation) THEN
			;
		END_IF
		
		// no change action
		
		//--------------------------------------------------------------------------------------
		// sub state machine for sequence
		CASE stSubSate.intState OF
			//--------------------------------------------------------------------------------------
			cCMD_INITIALIZED:
					// State Change Condition
					IF(TRUE) THEN
						stSubSate.intStateNext := cSTA_VER_Down;
					END_IF
					
			//--------------------------------------------------------------------------------------
			cSTA_VER_Down:
					pVER_CIF^.Job.intACmd := cCMD_EXTEND; // move to position down
					
					// State Change Condition
					IF (pVER_CIF^.Job.intState=cSTA_EXTEND) AND (pHOR_CIF^.Job.intState=cSTA_RETRACT) THEN // pick position
						stSubSate.intStateNext := cSTA_WAIT_Pick;
					ELSIF (pVER_CIF^.Job.intState=cSTA_EXTEND) THEN // place position
						stSubSate.intStateNext := cSTA_VER_Up;
					END_IF
					
			//--------------------------------------------------------------------------------------
			cSTA_WAIT_Pick:
	
					// State Change Condition
					IF(stSubSate.udiTimeInState_ms>=SIf.Par.udiWaitPick_ms) THEN
						stSubSate.intStateNext := cSTA_VER_Up;
					END_IF
					
			//--------------------------------------------------------------------------------------
			cSTA_VER_Up:
					pVER_CIF^.Job.intACmd := cCMD_RETRACT; // move to position up
					
					// State Change Condition
					IF (pVER_CIF^.Job.intState=cSTA_RETRACT) AND (pHOR_CIF^.Job.intState=cSTA_RETRACT) THEN // pick position
						stSubSate.intStateNext := cSTA_HOR_MoveToPlace;
					ELSIF (pVER_CIF^.Job.intState=cSTA_RETRACT) THEN // place position
						stSubSate.intStateNext := cSTA_HOR_MoveToPick;
					END_IF		
					
			//--------------------------------------------------------------------------------------
			cSTA_HOR_MoveToPlace:
					pHOR_CIF^.Job.intACmd := cCMD_EXTEND; // move to position place
					
					// State Change Condition
					IF(pHOR_CIF^.Job.intState=cSTA_EXTEND) THEN
						stSubSate.intStateNext := cSTA_VER_Down;
					END_IF
					
			//--------------------------------------------------------------------------------------
			cSTA_HOR_MoveToPick:
					pHOR_CIF^.Job.intACmd := cCMD_RETRACT; // move to position pick	
					
					// State Change Condition
					IF(pHOR_CIF^.Job.intState=cSTA_RETRACT) THEN
						stSubSate.intStateNext := cSTA_Finished;
					END_IF
			//--------------------------------------------------------------------------------------
			cSTA_Finished:
					;
					
		END_CASE
		stSubSate.intStateLastCycle := stSubSate.intState;
		IF (stSubSate.intState<>stSubSate.intStateNext) THEN
			stSubSate.intState := stSubSate.intStateNext;  // set next state for next cycle
			stSubSate.udiTimeInState_ms := 0; // reset timer
			// log state change -> open point
		ELSE
			// increment time in state	
			stSubSate.udiTimeInState_ms := stSubSate.udiTimeInState_ms + me.FUBInfo.udiSample_ms;
		END_IF
		
		
		

		// State Change Condition
		IF ((me.Alarm.eActivAlmClass=E_AlmClass.EOFF) OR (me.Alarm.eActivAlmClass=E_AlmClass.OFF)) THEN
			me.StateMachine.intStateNext := cSTA_OFFBusy;
		ELSIF(me.intCmd=cCMD_OFF) THEN
			me.StateMachine.intStateNext := cSTA_OFFBusy;
		ELSIF(me.intCmd=cCMD_INIT) THEN
			me.StateMachine.intStateNext := cSTA_INITBusy;
		ELSIF (stSubSate.intState=cSTA_Finished) THEN
			me.StateMachine.intStateNext := cSTA_RUN;
		END_IF
		stSubSate.strState := THIS^.getCmdState(intCmdState:=stSubSate.intState,bolState:=TRUE);
	END_IF




//--------------------------------------------------------------------------------------
// Exit action
	IF (me.StateMachine.intState<>me.StateMachine.intStateNext) THEN
		SIf.Cur.udiCycleTime_ms := me.StateMachine.udiTimeInState_ms;
		stSubSate.strState := '';
	END_IF
END_METHOD

METHOD PROTECTED sta_RUN : BOOL
// state implemetation
//--------------------------------------------------------------------------------------
// Entry action
	IF (me.StateMachine.intState<>me.StateMachine.intStateLastCycle) THEN
		me.StateMachine.intStateLastCycle := me.StateMachine.intState;
		bolfpCmd := FALSE; // reset flag positive edge of run command
	END_IF


//--------------------------------------------------------------------------------------
// Cyclic action
	IF (me.StateMachine.intState=me.StateMachine.intStateLastCycle) THEN

		// Simulation
		IF (CIf.SwCfg.bolSimulation) THEN
			;
		END_IF
		
		IF (bolfpCmd=FALSE) AND (me.intCmd<>cCMD_RUN) THEN
			bolfpCmd := TRUE;
		END_IF
		
		// State Change Condition
		IF ((me.Alarm.eActivAlmClass=E_AlmClass.EOFF) OR (me.Alarm.eActivAlmClass=E_AlmClass.OFF)) THEN
			me.StateMachine.intStateNext := cSTA_OFFBusy;
		ELSIF(me.intCmd=cCMD_OFF) THEN
			me.StateMachine.intStateNext := cSTA_OFFBusy;
		ELSIF(me.intCmd=cCMD_INIT) THEN
			me.StateMachine.intStateNext := cSTA_INITBusy;
		ELSIF (me.intCmd=cCMD_RUN) AND (bolfpCmd=TRUE) THEN // command RUN and positive flag command was onetime <> RUN
			me.StateMachine.intStateNext := cSTA_RUNBusy;
		END_IF
	END_IF




//--------------------------------------------------------------------------------------
// Exit action
	IF (me.StateMachine.intState<>me.StateMachine.intStateNext) THEN
		;
	END_IF
END_METHOD

METHOD PROTECTED CtrlInit : BOOL
SUPER^.CtrlInit();

// get child if
pHOR_CIF := p_fbHOR^.getCtrlCIf();
pVER_CIF := p_fbVER^.getCtrlCIf();

// set parent id
pHOR_CIF^.Info.intParentCtrlId := CIf.Info.intCtrlId;
pVER_CIF^.Info.intParentCtrlId := CIf.Info.intCtrlId;

//necessary???
THIS^.CIf.Info.p_aCIf[0] := THIS^.pHOR_CIF;
THIS^.CIf.Info.p_aCIf[1] := THIS^.pVER_CIF;
END_METHOD

METHOD checkChildAlmClass : BOOL
//------------------------------------------------------------------------------------------------------
// check child alarm classes
IF (pHOR_CIF^.Job.eMe_ActivAlmClass=E_AlmClass.EOFF) OR (pVER_CIF^.Job.eMe_ActivAlmClass=E_AlmClass.EOFF) THEN
	CIf.Job.eMe_ActivAlmClass := E_AlmClass.EOFF;
	me.Alarm.bolfp := TRUE;
ELSE
	IF (me.Alarm.bolfp) THEN
		CIf.Job.eMe_ActivAlmClass := E_AlmClass.NONE; // no reset necessary
		me.Alarm.bolfp := FALSE;
	END_IF
END_IF

//------------------------------------------------------------------------------------------------------
// set alarm class parent of childs
IF (CIf.Job.eParent_ActivAlmClass=E_AlmClass.EOFF) THEN
	pHOR_CIF^.Job.eParent_ActivAlmClass := CIf.Job.eParent_ActivAlmClass;
	pVER_CIF^.Job.eParent_ActivAlmClass := CIf.Job.eParent_ActivAlmClass;
ELSIF(CIf.Job.eMe_ActivAlmClass=E_AlmClass.EOFF) OR (CIf.Job.eMe_ActivAlmClass=E_AlmClass.OFF) THEN
	pHOR_CIF^.Job.eParent_ActivAlmClass := CIf.Job.eMe_ActivAlmClass;
	pVER_CIF^.Job.eParent_ActivAlmClass := CIf.Job.eMe_ActivAlmClass;
ELSE
	// no important alarm for child active
	pHOR_CIF^.Job.eParent_ActivAlmClass := E_AlmClass.NONE;
	pVER_CIF^.Job.eParent_ActivAlmClass := E_AlmClass.NONE;
END_IF
END_METHOD

METHOD PROTECTED getCmdState : STRING
VAR_INPUT
	intCmdState: INT;
	bolState: BOOL;
END_VAR
getCmdState := SUPER^.getCmdState(intCmdState:=intCmdState,bolState:=bolState); // get global/base defined cmds/states
IF (getCmdState='') THEN // global not defined get local
	// get string cmd/state string information in runtime
	IF (bolState=FALSE) THEN
		// cmd's
		//CASE intCmdState OF 
		//ELSE
				getCmdState := 'not defined';
		//END_CASE;
	ELSE
	
	// cmd's
		CASE intCmdState OF
			cSTA_VER_Down: 
				getCmdState := 'cSTA_VER_Down';
			cSTA_WAIT_Pick: 
				getCmdState := 'cSTA_WAIT_Pick';
			cSTA_HOR_MoveToPlace: 
				getCmdState := 'cSTA_HOR_MoveToPlace';
			cSTA_HOR_MoveToPick: 
				getCmdState := 'cSTA_HOR_MoveToPick';
			cSTA_Finished: 
				getCmdState := 'cSTA_Finished';
		END_CASE;
	END_IF
END_IF
END_METHOD

END_FUNCTION_BLOCK

// ---- POUs/Program/SlowPRG_1.TcPOU
PROGRAM SlowPRG_1
VAR
	bolPlcStartupDone: BOOL := FALSE;
	bolHostInitDone : BOOL := FALSE;
	bolInitDone : BOOL := FALSE;
	strInstance: STRING;
	pCtrl_CIf: POINTER TO T_Ctrl_CIf;
	intState: INT;
	bolSetCmd: BOOL;
END_VAR

(*__________________________________________________________________________________________________
¦	
¦	Vistaprint Schweiz GmbH
¦	CH - 8401 Winterthur
¦
¦	www.vistaprint.ch - info@vistaprint.ch
¦___________________________________________________________________________________________________

Function desription:
call of all controller (FUB) for the slow task class.


History:
Version		Date			Author		Comment
---------------------------------------------------------------------------------------------------
0.00.1		24.05.2013		AVME/KVO	Start history


___________________________________________________________________________________________________*)

// -----------------------------------------------------------------------------------------------
// Initialize the PLC Parameter and check the PLC health
// -----------------------------------------------------------------------------------------------
IF (NOT bolPlcStartupDone) THEN
	bolPlcStartupDone := TRUE;	
END_IF
// -----------------------------------------------------------------------------------------------


// -----------------------------------------------------------------------------------------------
// The host system is downloading all parameter at startup. 
// bolPlcStartupDone will be set to true after the Host is done with the initialization
// -----------------------------------------------------------------------------------------------
IF (bolPlcStartupDone AND (NOT bolHostInitDone) AND NOT bolInitDone) THEN
	bolHostInitDone := TRUE;
END_IF
// -----------------------------------------------------------------------------------------------


// -----------------------------------------------------------------------------------------------
// Start PLC code initialization
// -----------------------------------------------------------------------------------------------
IF NOT bolInitDone AND bolPlcStartupDone AND bolHostInitDone THEN
	
	// init	
	bolInitDone := TRUE;
END_IF
// -----------------------------------------------------------------------------------------------

// -----------------------------------------------------------------------------------------------
// Normal Run mode after all the initialization is done
// -----------------------------------------------------------------------------------------------
IF (bolInitDone AND bolPlcStartupDone AND bolHostInitDone) THEN
	
	//****************************************************************************************************
	// cyclic controller calls
	//****************************************************************************************************
	// call alarm message handler
	g_fbAlm_Man(intCtrlIdMax:=E_CtrlId.E_CtrlIdMax);
	
(* Tests
IF (g_a_pCtrlCIf[E_CtrlId.CYL_HOR2]<>0) AND bolSetCmd THEN // check pointer valid
	g_a_pCtrlCIf[E_CtrlId.CYL_HOR2]^.Job.intACmd := cCMD_EXTEND;
	bolSetCmd := FALSE;
END_IF;

IF (g_a_pCtrlInst[E_CtrlId.CYL_HOR2]<>0) THEN // check pointer valid
	pCtrl_CIf := g_a_pCtrlInst[E_CtrlId.CYL_HOR2]^.getCtrlCIf();
	intState:= pCtrl_CIf^.Job.intState;
END_IF;
*)
	
END_IF
// -----------------------------------------------------------------------------------------------

END_PROGRAM

// ---- POUs/Alarm/FB_Alm_Man.TcPOU
FUNCTION_BLOCK FB_Alm_Man
VAR_INPUT
	///max ctrl id in project defined
	intCtrlIdMax: INT;
END_VAR
VAR CONSTANT
	///config alarm handler
	c_uinMaxAlmElements: UINT := 99;
	///0: with history on PLC, auto clr
	c_uinModeAlarm: UINT := 1;
	///machine number 1
	c_udiMachineNr: UDINT := 1;
	// commands for the UI
	cCMD_RESET_ALL : INT := 2; // reset state=RST, reset state CLR
	cCMD_RESET_RST : INT  := 4; // reset state=RST, reset state CLR
	cCMD_RESET_CLR : INT  := 6; // reset state CLR -> c_uinModeAlarm = 1, automatic reset will be done on PLC
END_VAR
VAR
	//------------------------------------------------------------
	// UI interface
	// alarmarray PLC -> UI
	aAlm: ARRAY[0..c_uinMaxAlmElements] OF T_AlmElement;
	// command interface for UI -> PLC
	intAlmCmd: INT;
	
	//------------------------------------------------------------
	// real local variables
	fbGetLocalTime: NT_GetTime;
	strActTime: STRING;
	jj: UINT;
	EmptyAlmElement: T_AlmElement;
	intState: INT;
	intTestCtrl: INT := 12;
	intTestState: INT;
	udiTestAlarmNr: UDINT;
	dinTestInfo: DINT;
	aCtrlAlm: ARRAY[1..6] OF T_Ctrl_Alm;
	eActiveAlmClass: E_AlmClass;
END_VAR

(*__________________________________________________________________________________________________
¦	
¦	Vistaprint Schweiz GmbH
¦	CH - 8401 Winterthur
¦
¦	www.vistaprint.ch - info@vistaprint.ch
¦___________________________________________________________________________________________________

Function desription:
The alarm manager sets and clears alarms from the internal array. In the internal array all active 
alarms of a machine are listed. The list has no order. A new entry will be inserted at the next 
free place.


History:
Version		Date			Author		Comment
---------------------------------------------------------------------------------------------------
0.00.1		29.04.2013		AVME/KVO	Start history


___________________________________________________________________________________________________*)

// read out actual time
fbGetLocalTime.NETID := '';
fbGetLocalTime.START := NOT fbGetLocalTime.START;
fbGetLocalTime.TMOUT := T#5S;
fbGetLocalTime();
strActTime := TC2_UTILITIES.SYSTEMTIME_TO_STRING(fbGetLocalTime.TIMESTR); // yyyymmdd-HH:mm::ss

// interface for UI access
CASE intState OF
	
	0: // reset cmd
		intAlmCmd := cCMD_DONE; // Ready for new cmd
		intState := intState + 1;
		
	1: // wait for cmd
		IF (intAlmCmd=cCMD_RESET_ALL) OR (intAlmCmd=cCMD_RESET_CLR) OR  (intAlmCmd=cCMD_RESET_RST) THEN
			intState := intState + 1;
		END_IF
		
	2: // reset alarms
		// reset state=RST, reset state CLR
		THIS^.clearAlarm(((intAlmCmd=cCMD_RESET_ALL) OR (intAlmCmd=cCMD_RESET_RST)), TRUE);
		intState := intState + 1;
		
	3: // reset state machines
		FOR jj:=0 TO INT_TO_UINT(intCtrlIdMax) BY 1 DO
			IF (g_a_pCtrlCIf[jj]<>0) THEN // check if entry exist
				g_a_pCtrlCIf[jj]^.Job.bolAlmReset := TRUE;
			END_IF
		END_FOR
		intState := 0; // done

END_CASE



//**********************************************************************************************
// Test manual set/reset/clear alarm
//**********************************************************************************************
CASE intTestState OF
	
	0: // wait
		
	1: //CLR
		THIS^.setAlarm(intTestCtrl,udiTestAlarmNr,dinTestInfo,ADR(aCtrlAlm),E_AlmState.CLR,eActiveAlmClass);
		intTestState := 0;
		
	2: // RST
		THIS^.setAlarm(intTestCtrl,udiTestAlarmNr,dinTestInfo,ADR(aCtrlAlm),E_AlmState.RST,eActiveAlmClass);
		intTestState := 0;
		
	3: // SET
		THIS^.setAlarm(intTestCtrl,udiTestAlarmNr,dinTestInfo,ADR(aCtrlAlm),E_AlmState.SET,eActiveAlmClass);
		intTestState := 0;

END_CASE

METHOD setAlarm : E_AlmClass
VAR_INPUT
	///from controller 
	intCtrlId: INT;
	///local alarm number
	udiAlarmNr: UDINT;
	///additional information - string???
	dinInfo: DINT;
	///corresponding alarm class
	p_Ctrl_Alm: POINTER TO T_Ctrl_Alm;
	///clear, resetable
	intState: E_AlmState;
END_VAR
VAR_IN_OUT
	eMe_ActivAlmClass: E_AlmClass;
END_VAR
VAR
	InAlmElement: T_AlmElement;
	ii: UINT;
	uinEmptyIndex: UINT;
	bolEmptyIndexFound: BOOL;
	bolIndexUpdate: BOOL;
	p_LocCtrlAlm: POINTER TO T_Ctrl_Alm;
	e_LocAlmClass: E_AlmClass;
END_VAR
// entry/delete element
bolEmptyIndexFound := FALSE;

IF (p_Ctrl_Alm<>0) AND (udiAlarmNr>0) THEN // chack if pointer valid
	p_LocCtrlAlm := (p_Ctrl_Alm + (udiAlarmNr-1) * SIZEOF(T_Ctrl_Alm));
	e_LocAlmClass := p_LocCtrlAlm^.eAlmClass;
ELSE
	e_LocAlmClass := E_AlmClass.EOFF; // novalid pointer reached!!
END_IF


// check entry element
InAlmElement.udiMachineNr := c_udiMachineNr;
InAlmElement.intCtrlId := intCtrlId;
InAlmElement.udiAlarmNr := udiAlarmNr;
InAlmElement.udiNr := 100000*InAlmElement.udiMachineNr + INT_TO_UDINT(100*InAlmElement.intCtrlId) + InAlmElement.udiAlarmNr;
InAlmElement.dinInfo := dinInfo;
InAlmElement.eClass := e_LocAlmClass;
InAlmElement.intState := intState;
InAlmElement.strDTEntry := strActTime;

// loop over whole alarm array
FOR ii:= 0 TO c_uinMaxAlmElements BY 1 DO
	
	IF ((InAlmElement.intState=E_AlmState.SET) OR (InAlmElement.intState=E_AlmState.RST)) THEN 
		
		// search next empty element
		IF (bolEmptyIndexFound=FALSE) AND (aAlm[ii].udiNr=0) THEN
			uinEmptyIndex := ii;
			bolEmptyIndexFound := TRUE; // do new alarm element entry
		ELSIF(InAlmElement.udiNr = aAlm[ii].udiNr) THEN	// existing entry found
			bolIndexUpdate := TRUE;
			// refresh state, alarm additional info
			aAlm[ii].dinInfo := InAlmElement.dinInfo;
			aAlm[ii].intState := InAlmElement.intState;
			bolEmptyIndexFound := FALSE; // no new entry needed
			EXIT; // refresh done
		END_IF
		
	ELSIF (InAlmElement.intState=E_AlmState.CLR) THEN
		IF(InAlmElement.udiNr = aAlm[ii].udiNr) THEN	// existing entry found
			IF (c_uinModeAlarm=1) THEN // no history on PLC
				aAlm[ii] := EmptyAlmElement; // clear entry
			ELSE
				aAlm[ii].intState := E_AlmState.CLR; // set clear state -> entry in plc history if needed
			END_IF
			EXIT; // clear done
		END_IF
	END_IF
END_FOR

// Entry or refresh done and active alarm priority > allready active alarm class -> entry active alarm class
IF ((bolIndexUpdate) OR (bolEmptyIndexFound)) AND (InAlmElement.eClass>eMe_ActivAlmClass) THEN 
	eMe_ActivAlmClass := InAlmElement.eClass;
END_IF

// do new alarm element entry
IF (bolEmptyIndexFound) THEN
	IF ((InAlmElement.intState=E_AlmState.SET) OR (InAlmElement.intState=E_AlmState.RST)) THEN 
		aAlm[uinEmptyIndex] := InAlmElement;
	END_IF;
END_IF
END_METHOD

METHOD clearAlarm : BOOL
VAR_INPUT
	///-> clear all entries with state RST
	bolClear_RST: BOOL;
	///-> clear all entries with state CLR
	bolClear_CLR: BOOL;
END_VAR
VAR
	ii: UINT;
END_VAR

FOR ii:= 0 TO c_uinMaxAlmElements BY 1 DO
	
	IF (aAlm[ii].udiNr>0) THEN 
		
		IF (((aAlm[ii].intState=E_AlmState.RST) AND (bolClear_RST)) OR
			((aAlm[ii].intState=E_AlmState.CLR) AND (bolClear_CLR)))THEN
			
			aAlm[ii] := EmptyAlmElement; // clear entry
		END_IF
		
	END_IF
END_FOR
END_METHOD

END_FUNCTION_BLOCK
